// ---- POUs/Lib/Motion/CanOpenAxis/EcCoeSdo/EcCoeSdo_Par_Write_typ.TcDUT
TYPE EcCoeSdo_Par_Write_typ : 	
	STRUCT  (*parameter structure*)
		
        nSubIndex       : BYTE; 
        nIndex          : WORD;
        pSrcBuf         : POINTER TO DWORD; 
        cbBufLen        : UDINT; 
        tTimeout        : TIME := DEFAULT_ADS_TIMEOUT ;

	END_STRUCT
END_TYPE

// ---- POUs/Lib/Motion/CanOpenAxis/EcCoeSdo/EcCoeSdo_Status_typ.TcDUT
TYPE EcCoeSdo_Status_typ : 	
	STRUCT 
		Done : BOOL;
		Busy : BOOL;
		CommandAborted : BOOL;
		Active : BOOL ;
	END_STRUCT
END_TYPE

// ---- POUs/Lib/Motion/CanOpenAxis/eHomingMethods.TcDUT
{attribute 'qualified_only'}
{attribute 'strict'}
TYPE eHomingMethods :
(
	HarsrStopPosDir					:= -2,
	HarsrStopNegDir					:= -1,
	RlsAndIndexPulse 				:= 1,
	FlsAndIndexPulse 				:= 2,
	PositiveSwAndIndexPulse 		:= 3,
	ForwardOnPosSwAndIndexPulse 	:= 4,
	ForwardNegativeSwAndIndexPulse 	:= 5,
	ReverseNegativeSwAndIndexPulse 	:= 6,
	ReverseOnSwAndIndexPulse 		:= 7,
	ForwardOnSwAndIndexPulse 		:= 8,
	ReverseOnPosSwRLSAndIndexPulse	:= 9,
	ForwardOnNegSwAndIndexPulse 	:= 10,
	ForwardOnNegSwAndRLS		 	:= 11,
	ReverseOnPosFLSSwAndIndexPulse	:= 12,
	ForwardOnPosSwRlsAndIndexPulse 	:= 13,
	ReverseOnNegSwRlsAndIndexPulse 	:= 14,
	Reserve1						:= 15,
	Reserve2 						:= 16,
	RlsOnly							:= 17,
	FlsOnly							:= 18,
	ReverseOnNegSw				 	:= 19,
	ForwardOnPosSw					:= 20,
	ForwardOnNegSw					:= 21,
	ReverseOnPosSw				 	:= 22,
	ReverseOnNegFLS				 	:= 23,
	ForwardOnPosFLS					:= 24,
	ReverseOnPosFLS					:= 25,
	ForwardOnNegFLS					:= 26,
	ForwardOnNegRLS					:= 27,
	ReverseOnPosRLS					:= 28,
	ForwardOnPosRLS					:= 29,
	ReverseOnNegRLS					:= 30,
	Reserve3						:= 31,
	Reserve4 						:= 32,	
	IndexPulseNegDir   				:= 33,
	IndexPulsePosDir				:= 34,
	HomeAbs							:= 35,
	HomeCurrent						:= 37 
	
);
END_TYPE

// ---- POUs/Lib/Motion/CanOpenAxis/e_Homing_Contol_Word.TcDUT
{attribute 'qualified_only'}
{attribute 'strict'}
TYPE e_Homing_Contol_Word :
(
	SWITCH_ON 				:= 2#1,		
	Enable_VOLTAGE			:= 2#10,
	QUICK_STOP	 			:= 2#100 ,
	ENABLE_OPERATION		:= 2#1000 ,
	HOME_OPERATION_START	:= 2#10000 ,
	RESERVED1				:= 2#100000 ,
	RESERVED2				:= 2#1000000 ,
	FAULT_RESET				:= 2#10000000 ,
	HALT					:= 2#100000000
);
END_TYPE

// ---- POUs/Lib/Motion/CanOpenAxis/e_Homing_Status_Word.TcDUT
{attribute 'qualified_only'}
{attribute 'strict'}
TYPE e_Homing_Status_Word :
(
	READY_FOR_SWITCH_ON		:= 2#1,		
	SWITCHED_ON				:= 2#10,
	OPERATION_ENABLED		:= 2#100 ,
	FAULT					:= 2#1000 ,
	VOLTAGE_ENABLED			:= 2#10000 ,
	QUICK_STOP				:= 2#100000 , //5
	SWITCH_ON_DISABLED		:= 2#1000000 ,//6
	WARNING					:= 2#10000000 ,//7
	MANAFACTURE_SPECIFIC	:= 2#100000000,
	REMOTE					:= 2#1000000000,//9
	TARGET_REACHED			:= 2#10000000000,//10
	INTERNAL_LIMIT_ACTIVE   := 2#100000000000,//11
	HOMING_ATTAINED			:= 2#1000000000000,//12
	HOMING_ERROR			:= 2#10000000000000,//13	
	RESERVED				:= 2#100000000000000//14,15
);
END_TYPE

// ---- POUs/Lib/Motion/CanOpenAxis/Homing_CoE_Ctrl_Paramters_typ.TcDUT
TYPE Homing_CoE_Ctrl_Paramters_typ :
STRUCT
	HomingMethod  : SINT; 
	HomingSWSpeed : UDINT;
	HomingTrSpeed : UDINT; 
	HomingAcc     : UDINT;
	HomingOffset  : DINT;
 
END_STRUCT
END_TYPE

// ---- POUs/Lib/Motion/ErrorHandling_Lib/Eh_ErrorEntry_typ.TcDUT
TYPE Eh_ErrorEntry_typ:
STRUCT
	SourceId		: UDINT;
	SubSourceId		: UDINT;
	ErrorId			: UDINT;
	ErrorText		: STRING(500);
	MotorEvents		: enumMotorEvents;	
END_STRUCT
END_TYPE

// ---- POUs/Lib/Motion/EtherCAT/SDO_RW/Tc2_EtherCAT_typ/EcCoeSdoRead_CMD_typ.TcDUT
TYPE EcCoeSdoRead_CMD_typ :
	STRUCT
		Enable	: BOOL ;
	END_STRUCT
END_TYPE

// ---- POUs/Lib/Motion/EtherCAT/SDO_RW/Tc2_EtherCAT_typ/EcCoeSdoRead_Param_typ.TcDUT
TYPE EcCoeSdoRead_Param_typ :
	STRUCT
		sNetId          : T_AmsNetId; 
        nSlaveAddr      : UINT; 
        nSubIndex       : BYTE; 
        nIndex          : WORD;
		pDstBuf         : POINTER TO DWORD; 
		cbBufLen        : UDINT; 
		tTimeout        : TIME := DEFAULT_ADS_TIMEOUT; 
	END_STRUCT
END_TYPE

// ---- POUs/Lib/Motion/EtherCAT/SDO_RW/Tc2_EtherCAT_typ/EcCoeSdoRead_Status_typ.TcDUT
TYPE EcCoeSdoRead_Status_typ :
	STRUCT
		bBusy           : BOOL;
        bError          : BOOL;
	END_STRUCT
END_TYPE

// ---- POUs/Lib/Motion/EtherCAT/SDO_RW/Tc2_EtherCAT_typ/EcCoeSdoWrite_CMD_typ.TcDUT
TYPE EcCoeSdoWrite_CMD_typ :
	STRUCT
		Enable	: BOOL ;
	END_STRUCT
END_TYPE

// ---- POUs/Lib/Motion/EtherCAT/SDO_RW/Tc2_EtherCAT_typ/EcCoeSdoWrite_Param_typ.TcDUT
TYPE EcCoeSdoWrite_Param_typ :
	STRUCT
		sNetId          : T_AmsNetId; 
        nSlaveAddr      : UINT; 
        nSubIndex       : BYTE; 
        nIndex          : WORD;
        pSrcBuf         : POINTER TO DWORD; 
        cbBufLen        : UDINT; 
        //bExecute        : BOOL;
        tTimeout        : TIME := DEFAULT_ADS_TIMEOUT ;
	END_STRUCT
END_TYPE

// ---- POUs/Lib/Motion/EtherCAT/SDO_RW/Tc2_EtherCAT_typ/EcCoeSdoWrite_Status_typ.TcDUT
TYPE EcCoeSdoWrite_Status_typ :
	STRUCT
		bBusy           : BOOL;
        bError          : BOOL;
	END_STRUCT
END_TYPE

// ---- POUs/Lib/Motion/EtherCAT/SDO_RW/Tc2_EtherCAT_typ/EcSoeRead_CMD_typ.TcDUT
TYPE EcSoeRead_CMD_typ :
	STRUCT
		Enable	: BOOL ;
	END_STRUCT
END_TYPE

// ---- POUs/Lib/Motion/EtherCAT/SDO_RW/Tc2_EtherCAT_typ/EcSoeRead_Param_typ.TcDUT
TYPE EcSoeRead_Param_typ :
	STRUCT
		sNetId          : T_AmsNetId; 
        nSlaveAddr      : UINT; 
        nSubIndex       : BYTE; 
        nIdn            : WORD;
        nElement        : BYTE;
        nDriveNo        : BYTE;
        bCommand        : BOOL;
        pDstBuf         : POINTER TO DWORD; 
        cbBufLen        : UDINT; 
        bExecute        : BOOL;
        tTimeout        : TIME := DEFAULT_ADS_TIMEOUT;
	END_STRUCT
END_TYPE

// ---- POUs/Lib/Motion/EtherCAT/SDO_RW/Tc2_EtherCAT_typ/EcSoeRead_Status_typ.TcDUT
TYPE EcSoeRead_Status_typ :
	STRUCT
		bBusy           : BOOL;
        bError          : BOOL;
	END_STRUCT
END_TYPE

// ---- POUs/Lib/Motion/EtherCAT/SDO_RW/Tc2_EtherCAT_typ/EcSoeWrite_CMD_typ.TcDUT
TYPE EcSoeWrite_CMD_typ :
	STRUCT
		Enable	: BOOL ;
	END_STRUCT
END_TYPE

// ---- POUs/Lib/Motion/EtherCAT/SDO_RW/Tc2_EtherCAT_typ/EcSoeWrite_Param_typ.TcDUT
TYPE EcSoeWrite_Param_typ :
	STRUCT
		sNetId          : T_AmsNetId; 
        nSlaveAddr      : UINT; 
        nIdn            : WORD; 
        nElement        : BYTE;
        nDriveNo        : BYTE;
        pCommand        : BOOL;
        pSrcBuf         : POINTER TO DWORD; 
        cbBufLen        : UDINT; 
        bExecute        : BOOL;
        tTimeout        : TIME := DEFAULT_ADS_TIMEOUT; 
	END_STRUCT
END_TYPE

// ---- POUs/Lib/Motion/EtherCAT/SDO_RW/Tc2_EtherCAT_typ/EcSoeWrite_Status_typ.TcDUT
TYPE EcSoeWrite_Status_typ :
	STRUCT
		bBusy           : BOOL;
        bError          : BOOL;
	END_STRUCT
END_TYPE

// ---- POUs/Lib/Motion/EtherCAT/SDO_RW/Tc2_EtherCAT_typ/Tc2_EtherCAT_Command_axis_typ.TcDUT
TYPE Tc2_EtherCAT_Command_axis_typ : 	
	STRUCT  (*command structure*)
		EcCoeSdoWrite		: EcCoeSdoWrite_CMD_typ ;
		EcCoeSdoRead		: EcCoeSdoRead_CMD_typ ;
		EcSoeRead			: EcSoeRead_CMD_typ ;
		EcSoeWrite			: EcSoeWrite_CMD_typ ;
	END_STRUCT
END_TYPE

// ---- POUs/Lib/Motion/EtherCAT/SDO_RW/Tc2_EtherCAT_typ/Tc2_EtherCAT_Error_typ.TcDUT
TYPE Tc2_EtherCAT_Error_typ :
	STRUCT
		ErrorID : UDINT ;
		ErrorText : STRING[2048];
	END_STRUCT
END_TYPE

// ---- POUs/Lib/Motion/EtherCAT/SDO_RW/Tc2_EtherCAT_typ/Tc2_EtherCAT_Input_typ.TcDUT
TYPE Tc2_EtherCAT_Input_typ : 	
	STRUCT 
		Command 	: Tc2_EtherCAT_Command_axis_typ;
		Parameter 	: Tc2_EtherCAT_Parameter_axis_typ;
	END_STRUCT
END_TYPE

// ---- POUs/Lib/Motion/EtherCAT/SDO_RW/Tc2_EtherCAT_typ/Tc2_EtherCAT_Output_typ.TcDUT
TYPE Tc2_EtherCAT_Output_typ : 	
	STRUCT 
		Status 	: Tc2_EtherCAT_Statuses_typ;
		Error 	: Tc2_EtherCAT_Error_typ;
	END_STRUCT
END_TYPE

// ---- POUs/Lib/Motion/EtherCAT/SDO_RW/Tc2_EtherCAT_typ/Tc2_EtherCAT_Parameter_axis_typ.TcDUT
TYPE Tc2_EtherCAT_Parameter_axis_typ : 	
	STRUCT  (*parameter structure*)
		EcCoeSdoWrite		: EcCoeSdoWrite_Param_typ ;
		EcCoeSdoRead		: EcCoeSdoRead_Param_typ ;
		EcSoeRead			: EcSoeRead_Param_typ ;
		EcSoeWrite			: EcSoeWrite_Param_typ ;
	END_STRUCT
END_TYPE

// ---- POUs/Lib/Motion/EtherCAT/SDO_RW/Tc2_EtherCAT_typ/Tc2_EtherCAT_Statuses_typ.TcDUT
TYPE Tc2_EtherCAT_Statuses_typ :
	STRUCT
		EcCoeSdoWrite 	: EcCoeSdoWrite_Status_typ ;
		EcCoeSdoRead 	: EcCoeSdoRead_Status_typ ;
		EcSoeRead		: EcSoeRead_Status_typ ;
		EcSoeWrite		: EcSoeWrite_Status_typ ;
	END_STRUCT
END_TYPE

// ---- POUs/Lib/Motion/EtherCAT/SDO_RW/Tc2_EtherCAT_typ/Tc2_EtherCAT_typ.TcDUT
TYPE Tc2_EtherCAT_typ :
	STRUCT
		Input	: Tc2_EtherCAT_Input_typ ;
		Output	: Tc2_EtherCAT_Output_typ ;
	END_STRUCT
END_TYPE

// ---- POUs/Lib/Motion/External Libs/Data types/exCONSTANTS_MATH.TcDUT
TYPE exCONSTANTS_MATH :
STRUCT
	/// Kreiszahl PI 
	PI: REAL := 3.1415926535897931;
	/// PI * 2 
	PI2: REAL := 6.2831853071795862;
	/// PI * 4 
	PI4: REAL := 12.566370614359173;
	/// PI / 2 
	PI05: REAL := 1.5707963267949;
	/// PI / 4 
	PI025: REAL := 0.785398163397448;
	/// 1 / PI 
	PI_INV: REAL := 0.318309886183791;
	/// Euler constant e 
	E: REAL := 2.7182818284590451;
	/// 1 / e 
	E_INV: REAL := 0.367879441171442;
	/// Wurzel von 2 
	SQ2: REAL := 1.4142135623731;
	FACTS: ARRAY[0..12] OF DINT := [1, 1, 2, 6, 24, 120, 720, 5040, 40320, 362880, 3628800, 39916800, 479001600];
END_STRUCT
END_TYPE

// ---- POUs/Lib/Motion/External Libs/Data types/exCONSTANTS_PHYS.TcDUT
TYPE exCONSTANTS_PHYS :
STRUCT
	/// Lichtgeschwindigkeit in m/s 
	C: REAL := 299792458.0;
	/// elementarladung in Colomb = A * s 
	E: REAL := 1.60217653E-19;
	/// Erdbeschleunigung in m / s² 
	G: REAL := 9.80665;
	/// absoluter Nullpunkt in °C 
	T0: REAL := -273.15;
	/// Universelle Gaskonstante in J / (mol · K) 
	RU: REAL := 8.314472;
	/// NormalDruck in Pa 
	PN: REAL := 101325.0;
END_STRUCT
END_TYPE

// ---- POUs/Lib/Motion/FailureRport/Motor/enumFailReportControlFailures.TcDUT
//{attribute 'qualified_only'}
//{attribute 'strict'}
TYPE enumFailReportControlFailures :
(
	IllegalMessageReceived		:=0,
	FunctionBlockError	    	:=1,
	DriveNotReadyForCommand		:=2,
	IllegalParameterReceived	:=3,
	CycleTimeViolation			:=4,
	CommunicationErrorWithDrive	:=5,
	InternalTimeout 			:=6
);
END_TYPE

// ---- POUs/Lib/Motion/FailureRport/Motor/enumFailReportFailureType.TcDUT
//{attribute 'qualified_only'}
//{attribute 'strict'}
TYPE enumFailReportFailureType :
(
	NoFailure 			  :=0,
	MotorFailure 		  :=1,
	ControlFailure 		  :=2,
	CalibrationFailure	  :=3,
	PowerFailure		  :=4,
	FunctionalFailureHigh :=5,
	FunctionalFailureLow  :=6,
	ModuleFailure 		  :=8,
	GeneralDriveError	  :=9
);
END_TYPE

// ---- POUs/Lib/Motion/FailureRport/Motor/enumFailReportMotorFailures.TcDUT
//{attribute 'qualified_only'}
//{attribute 'strict'}
TYPE enumFailReportMotorFailures :
(
	PositionError 			:=0,
	SpeedError				:=1,
	HomeNotFound	 		:=2,
	OverCurrent				:=3,
	OverTemperature			:=4,
	FeedbackError		 	:=5,
	GeneralDriveError 		:=6
);
END_TYPE

// ---- POUs/Lib/Motion/FailureRport/Motor/enumFailReportSeverity.TcDUT
//{attribute 'qualified_only'}
//{attribute 'strict'}
TYPE enumFailReportSeverity :
(
	Warning 	:= 0,
	Error		:= 1,
	Critical	:= 2
	
);
END_TYPE

// ---- POUs/Lib/Motion/FailureRport/Motor/enumMotorEvents.TcDUT
{attribute 'qualified_only'}
{attribute 'strict'}
TYPE enumMotorEvents :
(
	NoEvents				:=0,
	MotorPositionError      :=1,
	MotorSpeedError	        :=2,
	MotorHomeNotFound	    :=3,
	MotorOverCurrent	    :=4,
	MotorOverTemp		    :=5,
	MotorFeedBackErr	    :=6,
	MotorGeneralError		:=7,
	MotorStalled			:=8,
	MotorSupplyError		:=9,
	PLCillegalMsg			:=10,
	PLCIllegalParam			:=11,
	DriveNotEnabled		    :=12,
	DriveNotReady           :=13,
	DriveComError           :=14,
	BreakResistorError      :=15
	
	

);
END_TYPE

// ---- POUs/Lib/Motion/FailureRport/Terminal/Group/Terminal_Group_Ctrl_typ.TcDUT
TYPE Terminal_Group_Ctrl_typ : 	
	STRUCT
  
		In : Terminal_Group_Input_typ;
		
		Out : Terminal_Group_Output_typ;
		
	END_STRUCT
END_TYPE

// ---- POUs/Lib/Motion/FailureRport/Terminal/Group/Terminal_Group_Input_typ.TcDUT
TYPE Terminal_Group_Input_typ : 	
	STRUCT 
		Par : Terminal_Group_Parameter_typ;
	END_STRUCT
END_TYPE

// ---- POUs/Lib/Motion/FailureRport/Terminal/Group/Terminal_Group_Monitor_typ.TcDUT
TYPE Terminal_Group_Monitor_typ : 	
	STRUCT  
		SubSysName		: STRING[20];	
	END_STRUCT
END_TYPE

// ---- POUs/Lib/Motion/FailureRport/Terminal/Group/Terminal_Group_Output_typ.TcDUT
TYPE Terminal_Group_Output_typ : 	
	STRUCT  
		Status:  Terminal_Group_Status_typ;
		Monitor: Terminal_Group_Monitor_typ;
	END_STRUCT
END_TYPE

// ---- POUs/Lib/Motion/FailureRport/Terminal/Group/Terminal_Group_Parameter_typ.TcDUT
TYPE Terminal_Group_Parameter_typ : 	
	STRUCT  (*parameter structure*)
		GroupName			: STRING[20];
		GroupID				: USINT;	
		PosForLog			: USINT;
	END_STRUCT
END_TYPE

// ---- POUs/Lib/Motion/FailureRport/Terminal/Group/Terminal_Group_Status_typ.TcDUT
TYPE Terminal_Group_Status_typ : 	
	STRUCT  		
		Active:         BOOL;	
		errorBit:       ULINT; 
		
	END_STRUCT
END_TYPE

// ---- POUs/Lib/Motion/FailureRport/Terminal/Terminal/Terminal_Ctrl_typ.TcDUT
TYPE Terminal_Ctrl_typ : 	
	STRUCT
  
		In : Terminal_Input_typ;
		
		Out : Terminal_Output_typ;
		
	END_STRUCT
END_TYPE

// ---- POUs/Lib/Motion/FailureRport/Terminal/Terminal/Terminal_Input_typ.TcDUT
TYPE Terminal_Input_typ : 	
	STRUCT 
		Par : Terminal_Parameter_typ;
	END_STRUCT
END_TYPE

// ---- POUs/Lib/Motion/FailureRport/Terminal/Terminal/Terminal_Monitor_typ.TcDUT
TYPE Terminal_Monitor_typ : 	
	STRUCT  
		SubSysName		: STRING[20];	
	END_STRUCT
END_TYPE

// ---- POUs/Lib/Motion/FailureRport/Terminal/Terminal/Terminal_Output_typ.TcDUT
TYPE Terminal_Output_typ : 	
	STRUCT  
		Status:  Terminal_Status_typ;
		Monitor: Terminal_Monitor_typ;
	END_STRUCT
END_TYPE

// ---- POUs/Lib/Motion/FailureRport/Terminal/Terminal/Terminal_Parameter_typ.TcDUT
TYPE Terminal_Parameter_typ : 	
	STRUCT  (*parameter structure*)
		Name				: STRING[30] :=  'Empty';
		ModuleID			: UINT;		
		PosForLog			: USINT;
	END_STRUCT
END_TYPE

// ---- POUs/Lib/Motion/FailureRport/Terminal/Terminal/Terminal_Status_typ.TcDUT
TYPE Terminal_Status_typ : 	
	STRUCT  
		TerminalState:  UDINT;
		Active:         BOOL;	
		Fault:          BOOL;
	END_STRUCT
END_TYPE

// ---- POUs/Lib/Motion/SercosAxis/SercosDrive_Ctrl_Adr_typ.TcDUT
TYPE SercosDrive_Ctrl_Adr_typ :
STRUCT
	//output
	ControlWord      : WORD;
	DriveError:       WORD;
	Diagnostic:       WORD;	
END_STRUCT
END_TYPE

// ---- POUs/Lib/ProgramBasic/LocalEvent_Typ.TcDUT
TYPE LocalEvent_Typ :
STRUCT
	EventHeader:EventHeader_Typ;
	EventParameters:EventParam_Typ;
	rEvent : REFERENCE TO EventHelper;
//	flowId:DINT;
END_STRUCT
END_TYPE

// ---- POUs/Lib/Signal/E_LutMode.TcDUT
{attribute 'qualified_only'}
{attribute 'strict'}
TYPE E_LutMode :
(
	eDisabled:= 0,
	ePhisicalToAnalog:= 1,
	eAnalogToPhisical:= 2
);
END_TYPE

// ---- POUs/Lib/Signal/ST_LookUpTableParam.TcDUT
TYPE ST_LookUpTableParam	 :
STRUCT
	arrPhisical:	ARRAY[0..40] OF LREAL;
	arrAnalog:		ARRAY[0..40] OF LINT;
	eLutMode:		E_LutMode;			
END_STRUCT
END_TYPE

// ---- POUs/Lib/System/CmdQueue/DUTs/DelayInfo_typ.TcDUT
TYPE DelayInfo_typ :
STRUCT	
	RequestId : UDINT;
	GroupId : UDINT;
	DelayType : eDelayType;
	DelayValue : ULINT; // ms or microns
	pExecuted : POINTER TO BOOL; // need to be persistant
	PrivateInfo : PVOID;
	Executed : BOOL;
	LagError : UDINT; // ms or microns
END_STRUCT
END_TYPE

// ---- POUs/Lib/System/CmdQueue/DUTs/eDelayType.TcTLEO
{attribute 'qualified_only'}
{attribute 'strict'}
TYPE eDelayType :
(
	Immediate := 0,
	DelayByTimer := 1,
	DelayByPos := 2
);
END_TYPE

// ---- GVLs/AxesList.TcGVL
//{attribute 'qualified_only'}
VAR_GLOBAL
	gWebAxes:		WebAxes_typ;	
END_VAR

// ---- GVLs/Consts.TcGVL
//{attribute 'qualified_only'}
VAR_GLOBAL CONSTANT
CONST_ZERO :DINT :=0;	





END_VAR

VAR_GLOBAL CONSTANT

// States		
	MACHINE_RUN_INIT:						INT:=0;
	MACHINE_GRIPPER_START_POSITION:			INT:=11;
	MACHINE_GRIPPER_EXCTRACT:				INT:=12;
	MACHINE_GRIPPER_OPEN:					INT:=13;
	MACHINE_GRIPPER_CLOSE:					INT:=14;
	MACHINE_GRIPPER_RETRACT:				INT:=15;
	
	MACHINE_GRIPPER_END_POSITION:			INT:=17;
	MACHINE_ENABLE_TENSION:					INT:=18;	
	//MACHINE_FRIPPER_WAIT_POSITION:			INT:=19;	
	
	MACHINE_WAIT_DANCER_FULL:				INT:=21;
	
	
	MACHINE_COLD_CUT_VALVE_OPEN:				INT:=10;
	MACHINE_WELD_VALVE_OPEN:					INT:=20;	
	MACHINE_HEATER_ON:							INT:=30;	
	MACHINE_HEATER_OFF:							INT:=40;
	MACHINE_VALVE_CLOSE:						INT:=50;	
	
	MACHINE_OUT_GRIPPER_START_POSITION:			INT:=60;
	MACHINE_OUT_GRIPPER_CLAMP:					INT:=61;
	MACHINE_OUT_GRIPPER_END_POSITION:			INT:=62;	
	
	MACHINE_CUT_WEB:							INT:=63;

	MACHINE_DONE:							INT:=100;	



END_VAR

// ---- GVLs/GVL.TcGVL
//{attribute 'qualified_only'}
VAR_GLOBAL
gMachineCtrl: Ctrl_Typ;
	
FB_Machine_Ctrl:FB_Machine_Ctrl;
FB_Machine_Run:FB_Machine_Run;
FB_Mechinit:FB_Mechinit;
FB_OFF:FB_OFF;
FB_Mechinit_Output:FB_MechinitOutput;

FB_RW_Ctrl:FB_RW_Ctrl;
RwInverter :FB_INV;


//WebHandling
	UW_1_AxisFB			: Beck5xxxAxis_FB;
	UW_1_MultiAxisFB	: MultiAxis_FB;
	UW_1_CyclicAxisFB	: CyclicAxis_FB;
	
	UW_2_AxisFB			: Beck5xxxAxis_FB;
	UW_2_MultiAxisFB	: MultiAxis_FB;
	UW_2_CyclicAxisFB	: CyclicAxis_FB;	
	
	Output_AxisFB		: ElmoBasicAxis_FB;
//	Uutput_MultiAxisFB	: MultiAxis_FB;
//	Uutput_CyclicAxisFB	: CyclicAxis_FB;
	
	UwVmaster_AxisFB		: CoE_BasicAxis_FB;
	
	//UW_MotorFailureReportFB 		: MotorFailureReport_FB;
	//UWMaster_MotorFailureReportFB 	: MotorFailureReport_FB;
	
END_VAR

// ---- GVLs/Persist.TcGVL
//{attribute 'qualified_only'}
VAR_GLOBAL  PERSISTENT 
    PersistentStruct:Persistent_Typ;
END_VAR

// ---- POUs/Lib/Logging/logLib/GVL_1.TcGVL
//{attribute 'qualified_only'}
VAR_GLOBAL CONSTANT
	MAX_COUNT_LOG_PARAM		: USINT := 5;	(*Maximum parameters index in log message variable data (from 0)*)
	LOCAL_ARRAY_LENGTH		: UINT := 32;	(* power oof 2 : The length of local (per task) array*)
	MAX_MEMBERS_TO_WRITE	: USINT := 8;
	GLOBAL_ARRAY_LENGTH		: UINT := 4*1024;(* power oof 2 : The length of global array*)
	LOG_TPL					: USINT := 0;
	LOG_MAIN_MOTOR			: USINT := 1;
	ENUM_OF_LAST_TASK		: USINT := 1;
	LOG_MSG_CATEGORY_LENGTH	: UINT := 10;
	LOG_MSG_TEXT_LENGTH		: USINT := 210;	(*The maximal length of log text *)
END_VAR

VAR_GLOBAL

END_VAR

// ---- POUs/Lib/Logging/PLC_ClientComm/UDP_Comm/PcComm/PcComm.TcGVL
//{attribute 'qualified_only'}
VAR_GLOBAL
	LogGlobalArray : LogGlobalArrayObj;	
END_VAR

// ---- POUs/Lib/Motion/External Libs/Global Variables/exConstants.TcGVL
{attribute 'Tc2GvlVarNames' := ''}
VAR_GLOBAL CONSTANT
	STRING_LENGTH: INT := 250;
	LIST_LENGTH: INT := 250;
END_VAR

// ---- POUs/Lib/Motion/External Libs/Global Variables/exGlobale_Variablen.TcGVL
{attribute 'Tc2GvlVarNames' := ''}
VAR_GLOBAL
	MATH: exCONSTANTS_MATH;
	PHYS: exCONSTANTS_PHYS;

END_VAR

// ---- POUs/MAIN.TcPOU
PROGRAM MAIN
VAR

init:BOOL;

uw1_Toque AT %I* 	: INT;
uw1_Position AT %I* 	: DINT;
TriggerOff:Trigger;
TriggerEM_Button:Trigger;

BuzzerTimer:TON;
END_VAR


IF init =FALSE THEN
	init:=TRUE;
	ACT_Init_param();
END_IF

ACT_Emergency();

ACT_IO();

ACT_fbCall();

ACT_Buzzer();

ACTION ACT_Buzzer:

BuzzerTimer.IN:= gMachineCtrl.IO.Out.PressDown OR gMachineCtrl.IO.Out.ColdCutPistonDown;
BuzzerTimer.PT:= T#3S;
BuzzerTimer();
IF gMachineCtrl.IO.Out.PressDown
AND  BuzzerTimer.Q = FALSE THEN
	gMachineCtrl.IO.Out.Buzzer := TRUE;
ELSE
	gMachineCtrl.IO.Out.Buzzer := FALSE;
END_IF
END_ACTION

ACTION ACT_Emergency:

IF gMachineCtrl.Cmd.EmStop THEN
	//FB_Machine_Ctrl.ResetCycle:=TRUE;
	//gMachineCtrl.Cmd.EmStop:=FALSE;
	
	gMachineCtrl.Cmd.SwitchOn:=FALSE;
END_IF
IF TriggerOff.EDGENEG(gMachineCtrl.Cmd.SwitchOn) THEN
	gMachineCtrl.Cmd.EmStop:=TRUE;
END_IF

IF TriggerEM_Button.EDGEPOS(gMachineCtrl.Cmd.EmStop) THEN
	gMachineCtrl.Cmd.EmStop:=TRUE;
END_IF
END_ACTION

ACTION ACT_fbCall:



RwInverter(
	//Set_Vel_Link:=gUVCtrl.Input.Par.UV_Inverter_Set_Speed , 
	//INV_Enable:=gUVCtrl.Input.Cmd.UV_Inverter_Run , 
	//HWlink:=gMachineCtrl.IO.RwInverter,
	ctrl:=gMachineCtrl.RwInverter,
	//ResetError:= , 
	MasterNetId:= , 
	nSlaveAddr:= , 
	nSubIndex:= , 
	nIndex:= , 
	//Actual_Vel_Link=>gUVCtrl.Output.Status.UV_Inverter_Actual_Speed , 
	Error=> , 
	ErrorCode=> , 
	Inv_Status=> );


	
FB_OFF.Ctrl_ref 			REF= gMachineCtrl;
FB_OFF.FB_Machine_Run_ref 	REF= FB_Machine_Run;
FB_OFF.FB_Mechinit_ref 		REF= FB_Mechinit;
FB_OFF();	
	
FB_Machine_Ctrl.Ctrl_ref 				REF= gMachineCtrl;
FB_Machine_Ctrl.FB_Machine_Run_ref 		REF= FB_Machine_Run;
FB_Machine_Ctrl.FB_Mechinit_ref 		REF= FB_Mechinit;
FB_Machine_Ctrl.FB_MechinitOutput_ref  	REF= FB_Mechinit_Output;
FB_Machine_Ctrl.FB_OFF_ref				REF= FB_OFF;
FB_Machine_Ctrl();

FB_Machine_Run.Ctrl_ref 		REF= gMachineCtrl;
FB_Machine_Run.FB_RW_Ctrl_ref	REF= FB_RW_Ctrl;
FB_Machine_Run();


FB_Mechinit.Ctrl_ref	REF= gMachineCtrl;
FB_Mechinit();


FB_Mechinit_Output.Ctrl_ref	REF= gMachineCtrl;
FB_Mechinit_Output();

//FB_RW_Ctrl.Ctrl_ref REF= gMachineCtrl;
//FB_RW_Ctrl();
END_ACTION

ACTION ACT_Init_param:

//	Dancer fill speed
gMachineCtrl.Parameters.DancerFillSpeed:= 90000;//[mil deg/sec]

gMachineCtrl.Parameters.NumberOfCycles:= 1;

//Motor Parmeters
//gMachineCtrl.Parameters.MotorVelocity:=600;//[rpm]
gMachineCtrl.Parameters.DistanceToMove:=1000;//[mm]


gMachineCtrl.Parameters.WebLinarSpeed:=350;//[mm/sec]
gMachineCtrl.Parameters.WebLinarSpeedSlow:=250;//[mm/sec]

gMachineCtrl.Parameters.UW_1_Param.ForcedDiameter:=400;//[mm/sec]
gMachineCtrl.Parameters.UW_2_Param.ForcedDiameter:=400;//[mm/sec]

gMachineCtrl.Parameters.UW_1_Param.SetTension := 150;
gMachineCtrl.Parameters.UW_2_Param.SetTension := 150;

gMachineCtrl.Parameters.UW_1_Param.kp:=0.1;
gMachineCtrl.Parameters.UW_1_Param.TN:=T#0MS;

gMachineCtrl.Parameters.UW_2_Param.kp:=0.1;
gMachineCtrl.Parameters.UW_2_Param.TN:=T#0MS;

gMachineCtrl.Parameters.UW_1_Param.kpMove:=1;
gMachineCtrl.Parameters.UW_1_Param.TNMove:=T#0MS;

gMachineCtrl.Parameters.UW_2_Param.kpMove:=1;
gMachineCtrl.Parameters.UW_2_Param.TNMove:=T#0MS;

//Output
gMachineCtrl.Parameters.OutGripperEndPosition :=1800;//mm
gMachineCtrl.Parameters.OutGripperHomeVelocity:=75;//mm
gMachineCtrl.Parameters.OutGripperProcessVelocity:=1000;//mm
END_ACTION

ACTION ACT_IO:


//IO
gMachineCtrl.IO.In.PrimeryPressFeedback(
	SimFlag:= gMachineCtrl.Simulation);
	
gMachineCtrl.IO.In.SeconderyPressFeedbak(
	SimFlag:= gMachineCtrl.Simulation);
	
gMachineCtrl.IO.In.E_StopPressed := NOT(gMachineCtrl.IO.In.E_StopPressedRaw);

gMachineCtrl.IO.In.UW_1_DancerFull :=NOT( gMachineCtrl.IO.In.UW_1_DancerFullRaw);
gMachineCtrl.IO.In.UW_2_DancerFull :=NOT( gMachineCtrl.IO.In.UW_2_DancerFullRaw);	

gMachineCtrl.IO.In.UW_1_DancerEmpety :=NOT( gMachineCtrl.IO.In.UW_1_DancerEmpetyRaw);
gMachineCtrl.IO.In.UW_2_DancerEmpety :=NOT( gMachineCtrl.IO.In.UW_2_DancerEmpetyRaw);	

gMachineCtrl.IO.Out.Output_GripperOpen:= NOT (gMachineCtrl.IO.Out.Output_GripperClose);
END_ACTION

END_PROGRAM

// ---- POUs/Lib/Trigger.TcPOU
FUNCTION_BLOCK FINAL Trigger
VAR_INPUT
END_VAR
VAR_OUTPUT
END_VAR
VAR
	rTrig : R_TRIG ;
	ftrig : F_TRIG ;
END_VAR

METHOD PUBLIC EDGENEG : BOOL
VAR_INPUT
	input : BOOL ;
END_VAR

fTrig.CLK := input ;
fTrig();

EDGENEG := fTrig.Q ;
END_METHOD

METHOD PUBLIC EDGEPOS : BOOL
VAR_INPUT
	input : BOOL ;
END_VAR

rTrig.CLK := input ;
rTrig();

EDGEPOS := rTrig.Q ;
END_METHOD

METHOD ONE_SHOT : BOOL
VAR_INPUT
	input : BOOL ;
END_VAR
rTrig.CLK := input ;
rTrig();

fTrig.CLK := input ;
fTrig();

ONE_SHOT := rTrig.Q OR fTrig.Q;
END_METHOD

END_FUNCTION_BLOCK

// ---- POUs/App/FB_OFF.TcPOU
FUNCTION_BLOCK FB_OFF EXTENDS CycleHandleFB
VAR_INPUT
	Ctrl_ref:			REFERENCE TO Ctrl_Typ;
	FB_RW_Ctrl_ref:			REFERENCE TO FB_RW_Ctrl;
	FB_Machine_Run_ref:		REFERENCE TO FB_Machine_Run;
	FB_Mechinit_ref:		REFERENCE TO FB_Mechinit;

	
END_VAR
VAR_OUTPUT
END_VAR
VAR
	MethInitDone:		BOOL;
END_VAR

VAR CONSTANT
// States are global
		
	OFF_INIT:			INT:=0;
	OFF_STOP_MOTOR:		INT:=5;
	OFF_GEAR_OUT:		INT:=6;
	OFF_MOTOR:			INT:=10;
	OFF_RESET_CYCLES:	INT:=20;
	OFF_RESET_IO:	INT:=30;
	OFF_DONE:			INT:=100;
END_VAR



IF NOT MethInitDone THEN
	MethInitDone	:= Meth_Init();
END_IF

IF  THIS^.CMD.Pause = FALSE THEN
	
	//-----------------------------
	//State Machine
	//-----------------------------
	CASE THIS^.StepNo OF
		OFF_INIT:
			IF THIS^.StepOneShotTrig THEN
				THIS^.Monitoring.StepMessage	:= 'Init: Start.';
				THIS^.Delay(IN:=FALSE);
			ELSIF Meth_Enable(TRUE) THEN
				THIS^.StepNo	:= 	OFF_RESET_IO;
			END_IF
			
			OFF_RESET_IO:
				IF THIS^.StepOneShotTrig THEN
					THIS^.Monitoring.StepMessage	:= 'Rest all IO';
				ELSIF Meth_Rest_IO() THEN
					THIS^.StepNo	:= 	OFF_GEAR_OUT;
				END_IF			
			
			OFF_GEAR_OUT:
				IF THIS^.StepOneShotTrig THEN
					THIS^.Monitoring.StepMessage	:= 'Gear Out';
					THIS^.Meth_GearOut(FALSE);
				ELSIF Meth_GearOut(TRUE) THEN
					THIS^.StepNo	:= 	OFF_STOP_MOTOR;
				END_IF					
				
			OFF_STOP_MOTOR:
				IF THIS^.StepOneShotTrig THEN
					THIS^.Monitoring.StepMessage	:= 'Stop Motors';
					THIS^.Meth_StopMotors(FALSE);
				ELSIF Meth_StopMotors(TRUE) THEN
					THIS^.StepNo	:= 	OFF_MOTOR;
				END_IF					
				
			OFF_MOTOR:
				IF THIS^.StepOneShotTrig THEN
					THIS^.Monitoring.StepMessage	:= 'Switch Motors Off';
					THIS^.Meth_SwitchOff(FALSE);
				ELSIF Meth_SwitchOff(TRUE) THEN
					THIS^.StepNo	:= 	OFF_RESET_CYCLES;
				END_IF		

			OFF_RESET_CYCLES:
				IF THIS^.StepOneShotTrig THEN
					THIS^.Monitoring.StepMessage	:= 'Rest all cycles';
				ELSIF Meth_ResatAllCycles() THEN
					THIS^.StepNo	:= 	OFF_DONE;
				END_IF				
				
					
				
			OFF_DONE:
				IF THIS^.StepOneShotTrig THEN
					THIS^.Monitoring.StepMessage	:= 'OFF cycle Done';
				ELSIF Meth_Done(TRUE) THEN
					THIS^.StepNo	:= 	OFF_INIT;
				END_IF					
				
		END_CASE
	
	ELSE
		THIS^.Monitoring.StepMessage:= 'Pause';
		
		IF THIS^.Status.Fault = TRUE THEN
		//IF Meth_EmStop(TRUE) THEN
				THIS^.CMD.ResetCycle	:= TRUE;		// Reset the all state machine to start point
		//END_IF
			
		END_IF
		
	END_IF
	
	THIS^.Delay();
	THIS^.CH_Logic();
	
	// Reset Meth_EmStop when at Init State
	IF THIS^.Pause = FALSE THEN
		//Meth_EmStop(FALSE);
	END_IF

METHOD PRIVATE Meth_Done : BOOL
VAR_INPUT
	Execute: 	BOOL;
END_VAR


	//THIS^.Monitoring.StepMessage			:= 'Press 1 engage';
	//THIS^.Monitoring.Error_Text				:= 'Press 1 engage Fail';
	//THIS^.CMD.Deacivate_Sequence_Time_Out	:= TRUE;	// Disable time out to the all sequence
	//THIS^.CMD.DeactivateStepTimeOut			:= TRUE;	// Disable time out to the actual step
	//THIS^.Parameter.TimeOut					:= T#5S;

	THIS^.Status.Done		:= TRUE;
	THIS^.Status.Running	:= FALSE;									
	Meth_Done	:= TRUE;
END_METHOD

METHOD PRIVATE Meth_Enable : BOOL
VAR_INPUT
	Execute: 	BOOL;
END_VAR


IF THIS^.CMD.Start THEN
	
	THIS^.Monitoring.StepMessage			:= 'Start';
	THIS^.Monitoring.Error_Text				:= 'Start Fail';
	THIS^.CMD.Deacivate_Sequence_Time_Out	:= TRUE;	// Disable time out to the all sequence
	THIS^.CMD.DeactivateStepTimeOut			:= TRUE;	// Disable time out to the actual step
	THIS^.Parameter.TimeOut					:= T#0.5S;

	THIS^.CMD.Start			:= FALSE;
	THIS^.Status.Done		:= FALSE;
	THIS^.Status.Running	:= TRUE;
	
	// Reset Commands and Statuses												
	
	Meth_Enable	:= TRUE;
END_IF
END_METHOD

METHOD Meth_GearOut : BOOL
VAR_INPUT
	Execute: 	BOOL;
END_VAR
VAR_INST	
	ExecuteTrig: 	Trigger;	
END_VAR
IF ExecuteTrig.EDGEPOS(Execute) THEN
	Meth_GearOut	:= FALSE;
	THIS^.SubStepNo:= 	1;	
END_IF

IF ExecuteTrig.EDGENEG(Execute) THEN
	Meth_GearOut	:=	FALSE;
END_IF

CASE THIS^.SubStepNo OF
	   
	1:
	
		IF (gWebAxes.UW_1.Crtl.Basic_axis.Output.Status.AxisStatus.SynchronizedMotion = TRUE) THEN
			THIS^.Monitoring.StepMessage	:= 'Set Gear out command UW1';							
			gWebAxes.UW_1.Crtl.MultiAxis.Input.Command.GearInMultiMaster.DisengageSlave	:= TRUE;
			THIS^.SubStepNo	:= 2;	
		ELSE
			THIS^.Monitoring.StepMessage	:= 'UW1 not synchronized, continue';	
			THIS^.SubStepNo	:= 2;				
		END_IF	
			
	
	2:	
		IF (gWebAxes.UW_2.Crtl.Basic_axis.Output.Status.AxisStatus.SynchronizedMotion = TRUE) THEN
			THIS^.Monitoring.StepMessage	:= 'Set Gear out command UW2';							
			gWebAxes.UW_2.Crtl.MultiAxis.Input.Command.GearInMultiMaster.DisengageSlave	:= TRUE;
			THIS^.SubStepNo	:= 3;	
		ELSE
			THIS^.Monitoring.StepMessage	:= 'UW2 not synchronized, continue';	
			THIS^.SubStepNo	:= 3;				
		END_IF	
		
	3:	
		THIS^.Monitoring.StepMessage:= 'Wait for Gear out UW 1+2';
									
		IF  gWebAxes.UW_1.Crtl.Basic_axis.Output.Status.AxisStatus.SynchronizedMotion = FALSE
		AND gWebAxes.UW_2.Crtl.Basic_axis.Output.Status.AxisStatus.SynchronizedMotion = FALSE THEN
			Meth_GearOut:=TRUE;
		END_IF	

							
END_CASE
END_METHOD

METHOD Meth_Init :BOOL
VAR_INPUT
END_VAR
//resets


Meth_Init:=TRUE;
END_METHOD

METHOD Meth_ResatAllCycles : BOOL
VAR_INPUT
END_VAR

FB_Machine_Run_ref.ResetCycle	 :=TRUE;
FB_Mechinit_ref.ResetCycle		 :=TRUE;


Meth_ResatAllCycles:=TRUE;
END_METHOD

METHOD Meth_Rest_IO : BOOL
VAR_INPUT
	
END_VAR

Ctrl_ref.IO.Out.HeaterOn := FALSE;
gMachineCtrl.IO.Out.GripperRetract:=FALSE;
gMachineCtrl.IO.Out.GripperOpen:=FALSE;

gMachineCtrl.IO.Out.ExternalNipMotor:=FALSE;

gMachineCtrl.IO.Out.Output_GripperClose:=FALSE;

gMachineCtrl.IO.Out.Buzzer	:=FALSE;

gMachineCtrl.IO.Out.ColdCutPistonDown:=FALSE;	

Meth_Rest_IO:=TRUE;
END_METHOD

METHOD Meth_StopMotors : BOOL
VAR_INPUT
	Execute: 	BOOL;
END_VAR
VAR_INST	
	ExecuteTrig: 	Trigger;	
END_VAR
IF ExecuteTrig.EDGEPOS(Execute) THEN
	Meth_StopMotors	:= FALSE;
	THIS^.SubStepNo:= 	1;	
END_IF

IF ExecuteTrig.EDGENEG(Execute) THEN
	Meth_StopMotors	:=	FALSE;
END_IF

CASE THIS^.SubStepNo OF
	   
	1:
		THIS^.Monitoring.StepMessage:= 'Stop Motors';
		
		gWebAxes.UW_1.Crtl.Basic_axis.Input.Parameter.Acceleration := 	10000000;
		gWebAxes.UW_1.Crtl.Basic_axis.Input.Parameter.Deceleration := 	10000000;		
		gWebAxes.UW_1.Crtl.Basic_axis.Input.Command.Stop :=		TRUE;
		
		gWebAxes.UW_2.Crtl.Basic_axis.Input.Parameter.Acceleration := 	10000000;
		gWebAxes.UW_2.Crtl.Basic_axis.Input.Parameter.Deceleration := 	10000000;		
		gWebAxes.UW_2.Crtl.Basic_axis.Input.Command.Stop :=		TRUE;		
		
		gWebAxes.Output.Crtl.Basic_axis.Input.Parameter.Acceleration := 	10000;//[mm
		gWebAxes.Output.Crtl.Basic_axis.Input.Parameter.Deceleration := 	10000;		
		gWebAxes.Output.Crtl.Basic_axis.Input.Command.Stop :=		TRUE;		
						
				
								
		THIS^.SubStepNo	:= 2;		
			
	
	2:	
		THIS^.Monitoring.StepMessage:= 'Wait for standstill UW 1';
									
		IF gWebAxes.UW_1.Crtl.Basic_axis.Output.Status.AxisStatus.StandStill
		OR gWebAxes.UW_1.Crtl.Basic_axis.Output.Status.AxisStatus.Disabled THEN
			THIS^.SubStepNo	:= 3 ;
		END_IF
		
	3:	
		THIS^.Monitoring.StepMessage:= 'Wait for standstill UW 2';
									
		IF gWebAxes.UW_1.Crtl.Basic_axis.Output.Status.AxisStatus.StandStill
		OR  gWebAxes.UW_2.Crtl.Basic_axis.Output.Status.AxisStatus.Disabled THEN
			THIS^.SubStepNo	:= 4 ;
		END_IF	

	4:	
		THIS^.Monitoring.StepMessage:= 'Wait for standstill Output';
									
		IF gWebAxes.Output.Crtl.Basic_axis.Output.Status.AxisStatus.StandStill
		OR  gWebAxes.Output.Crtl.Basic_axis.Output.Status.AxisStatus.Disabled THEN
			//THIS^.SubStepNo	:= 4 ;
			Meth_StopMotors:=TRUE;
		END_IF								
END_CASE
END_METHOD

METHOD Meth_SwitchOff : BOOL
VAR_INPUT
	Execute: 	BOOL;
END_VAR
VAR_INST
	ExecuteTrig: 	Trigger;
END_VAR


IF ExecuteTrig.EDGEPOS(Execute) THEN
	Meth_SwitchOff:=	FALSE;
	THIS^.SubStepNo:= 	1;	
END_IF

IF ExecuteTrig.EDGENEG(Execute) THEN
	Meth_SwitchOff:=	FALSE;
END_IF

CASE THIS^.SubStepNo OF
	(* Power ON*)
	1:
		THIS^.Monitoring.StepMessage	:= 'Power OFF';								
		gWebAxes.UW_1.Crtl.Basic_axis.Input.Command.Power		:= FALSE;
		gWebAxes.UW_2.Crtl.Basic_axis.Input.Command.Power		:= FALSE;	
		gWebAxes.Output.Crtl.Basic_axis.Input.Command.Power		:= FALSE;
		
		THIS^.SubStepNo:= 2;		
	
	2:	
		THIS^.Monitoring.StepMessage:= 'Wait for Disabled UW 1';
									
		IF gWebAxes.UW_1.Crtl.Basic_axis.Output.Status.AxisStatus.Disabled THEN
			THIS^.SubStepNo	:= 3 ;
		END_IF
		
	3:	
		THIS^.Monitoring.StepMessage:= 'Wait for Disabled UW 2';
									
		IF gWebAxes.UW_2.Crtl.Basic_axis.Output.Status.AxisStatus.Disabled  THEN
			THIS^.SubStepNo	:= 4 ;
		END_IF	
	4:	
		THIS^.Monitoring.StepMessage:= 'Wait for Disabled Output';
									
		IF gWebAxes.Output.Crtl.Basic_axis.Output.Status.AxisStatus.Disabled  THEN
			Meth_SwitchOff	:= TRUE;
		END_IF		
		
							
END_CASE
END_METHOD

END_FUNCTION_BLOCK

// ---- POUs/Lib/CH Obj/CycleHandleFB.TcPOU
FUNCTION_BLOCK  CycleHandleFB 
VAR_IN_OUT

END_VAR

VAR_INPUT
	//pFlowID: 			POINTER TO DINT :=ADR(DummyFlowID) ;
	SetEvent:			BOOL;
		
END_VAR
VAR_OUTPUT
	//Error 				: Error_Handler_typ;
END_VAR
VAR 
	// ErrorReportStruct 	:  FailureReport_Typ;	

	CMD					: Basic_cycle_CMD_typ ;
	Monitoring			: Basic_cycle_Mon_typ ;
	Status				: Basic_cycle_Status_typ ;
	Parameter			: Basic_cycle_Param_typ ;
	AtReady				: BOOL;
	Delay 				: TON ;
	StepOneShotTrig		: BOOL;
	LogMsg_0 			: LogMsg ;
	//fbClearFaultHandler_0 : fbClearFaultHandler;
	ResetError 			: R_TRIG;
	rTrigCycleDone 		: R_TRIG;
	fTrigCycleRunning 	: F_TRIG;
	rTrigCycleStart		: R_TRIG;	
	Init_trig 			: R_TRIG;
	ResetFaultTrig 		: R_TRIG;
	ResetAllTrig 		: R_TRIG;
	ResumeAllTrig 		: R_TRIG;
	LastStepMessage 	: STRING[100];
	LastStepNo 			: DINT;
	LastSubStepNo		: DINT ;
	TimeOutFault		: BOOL;
	CycleTIME 			: TON;
	StepTimerTOut 		: TON;
	SubStepTimerTOut 	: TON;
	ErrorAcknowledge 	: BOOL;
	Triger1 			: Trigger ;
	Triger2 			: Trigger ;
	Triger3 			: Trigger ;
	Triger4 			: Trigger ; 
	Triger5 			: Trigger ; 

	DummyFlowID			: DINT :=0;
	//fbCHPrgmBasic 		: FB_PrgmBasic;

	//rEvent : 			REFERENCE TO EventHelper;
	//EventHeader:		EventHeader_Typ;
	//EventParameters:	EventParam_Typ;	
END_VAR

METHOD PROTECTED CH_Logic : BOOL
VAR_STAT
	EventSent: 			BOOL;
END_VAR
VAR
	stenNomForLog	: DINT;
END_VAR

	IF CMD.LogMsgInit THEN      
		CMD.LogMsgInit := FALSE ;
		fnLogMsgInit(ADR(LogMsg_0), Parameter.ThreadName, ADR(LogGlobalArray), ADR(Parameter.PosForLog));
		LogMsg_0.Enable:= 		TRUE;
		CMD.EnableStateLogging:= TRUE;
		Parameter.ExternalLogType := LOG_INFO ;
	END_IF

	// Write state name for every change of Step Message
	IF (Monitoring.StepMessage) <> (LastStepMessage) THEN
		LastStepMessage := Monitoring.StepMessage ;
		// fnLogMsg(ADR(LogMsg_0), LOG_INFO, CONCAT(CONCAT(Parameter.CHName,', State = %d, FlowID = %d '),Monitoring.StepMessage),LastStepNo,pFlowID^,0);	
		IF CMD.EnableStateLogging THEN
			IF (Parameter.StepMessageIsForNewState) THEN
				Parameter.StepMessageIsForNewState	:= FALSE;
				stenNomForLog	:= StepNo;
			ELSE
				stenNomForLog	:= LastStepNo;
			END_IF
			fnLogMsg(ADR(LogMsg_0), LOG_INFO, CONCAT(CONCAT(CONCAT(Parameter.CHName, ', '),Monitoring.StepMessage),', State = %d.'), stenNomForLog,0,0);	
		END_IF
	END_IF
	
	

				
	//Update Step Num for Visu
	IF Triger1.EDGEPOS(Monitoring.LastStep <> Monitoring.StepNo) THEN 
		Monitoring.Visu_StepNo := LastStepNo ;
	ELSIF Status.CycleStuck AND NOT CMD.Pause THEN
		Monitoring.Visu_StepNo := Monitoring.StepNo ;
	ELSIF (Monitoring.StepNo = 0)THEN
		Monitoring.Visu_StepNo := 0 ;
	END_IF
	
	
	rTrigCycleStart(CLK:= CMD.Start);	
	IF rTrigCycleStart.Q AND Status.Running AND Monitoring.StepNo > 0 THEN
		CMD.Start:=	FALSE;		
		fnLogMsg(ADR(LogMsg_0), LOG_ERROR, CONCAT(Parameter.CHName ,' ,Start Command While Cycle Running was ignored, FlowID = %d'),0,0,0);
	END_IF

	
	(*************************** Step By Step *****************************************)
	// Step By Step Logic: If Step By Step bit set:
	//							- We stay at the same step 
	//							- We set the Pause flag
	//							- We whait for Resume bit to set to continue
	(********************************************************************)
	IF CMD.StepByStep AND (CMD.Resume OR ResumeAllTrig.Q) THEN
		CMD.Resume	:=FALSE;
		CMD.Pause	:=FALSE;
	END_IF

	IF (CMD.StepByStep AND LastStepNo <> Monitoring.StepNo)THEN
		CMD.Pause	:=TRUE;
	END_IF

	rTrigCycleDone(CLK := Status.Done);
	IF CMD.StepByStep AND rTrigCycleDone.Q THEN
		CMD.Pause	:=FALSE;
	END_IF

	(*************************** Step Time Out *****************************************)
	// Time Out Logic: If timeout elapsed:
	//							- We set the FAULT flag
	//							- We set the Error_Number and Error_Text
	//							- We set the Pause flag
	(********************************************************************)
	
	//SubStep Stuck
	Status.SubStepStuck :=  (Monitoring.SubStepNo = LastSubStepNo) AND (Status.Running) AND (Monitoring.SubStepNo <> 0);
	LastSubStepNo := Monitoring.SubStepNo;
	
	SubStepTimerTOut.PT := Parameter.TimeOut ;
	SubStepTimerTOut.IN := Status.SubStepStuck
							AND NOT CMD.Pause
							AND NOT CMD.DeactivateStepTimeOut ;
					
	SubStepTimerTOut();
	Monitoring.SubStep_TimeOut := SubStepTimerTOut.ET ;

	//Step Stuck
	Status.CycleStuck:= (LastStepNo = Monitoring.StepNo)
			 AND (Status.Running) 
			 AND Monitoring.SubStepNo = 0 ;
			
	
	StepTimerTOut.PT := Parameter.TimeOut ;
	StepTimerTOut.IN := Status.CycleStuck
							AND NOT CMD.Pause
							AND NOT CMD.StepByStep
							AND NOT CMD.DeactivateStepTimeOut ;					
	StepTimerTOut();

	Monitoring.Step_TimeOut := StepTimerTOut.ET ;
	
	
	IF StepTimerTOut.Q OR SubStepTimerTOut.Q OR SetEvent THEN
		SetEvent := FALSE ;
		Status.Fault:=	TRUE;
		TimeOutFault:=	TRUE;
	END_IF
	
		 
	IF Status.Fault THEN
		CMD.Pause := TRUE;
	END_IF

	// Logging & Event
	IF Triger2.EDGEPOS(Status.Fault) THEN
		IF TimeOutFault THEN
			IF 	Monitoring.Error_Text = Monitoring.StepMessage THEN
				fnLogMsg(ADR(LogMsg_0),
				 LOG_ERROR,
					CONCAT(
						CONCAT(
							CONCAT(Parameter.CHName,', State = %d ,SubState = %d, FlowID = %d,'),
																					Monitoring.Error_Text),
																					' ,Fault - Time Out Elaspsed'),
																						Monitoring.StepNo,
																						Monitoring.SubStepNo,0);
			ELSE
				fnLogMsg(ADR(LogMsg_0),
				 LOG_ERROR,
					CONCAT(
						CONCAT(
							CONCAT(Parameter.CHName,', State = %d ,SubState = %d, FlowID = %d,'),
																					Monitoring.Error_Text),
																					' Fault - By Event'),
																						Monitoring.StepNo,
																						Monitoring.SubStepNo,0);
			END_IF	

		//	IF NOT __ISVALIDREF(rEvent) THEN
		//		//rEvent REF=	ev_PLC_INTERNAL_TIMEOUT;	
		//		Monitoring.ExternalLogText := 'No Link to Event, send default PLC internal Timeout event';
		//		CMD.WriteExternalFaultLogCMD := TRUE;
		//	END_IF
			//fbCHPrgmBasic.mEventThrow(rEvent,ADR(EventHeader),ADR(EventParameters));
				
		ELSE
			
			fnLogMsg(ADR(LogMsg_0),
			 LOG_ERROR,
				CONCAT(
					CONCAT(
						CONCAT(Parameter.CHName,', State = %d ,SubState = %d, FlowID = %d ,'),
																				Monitoring.Error_Text),
																				' Fault - By External Event'),
																					Monitoring.StepNo,
																					Monitoring.SubStepNo,0);
		
			//Event Parames reset
			//memset(ADR(EventParameters),0,SIZEOF(EventParameters)) ;
		END_IF
		
		
	END_IF
	
	IF CMD.WriteExternalFaultLogCMD THEN
		CMD.WriteExternalFaultLogCMD := FALSE ;
		fnLogMsg(ADR(LogMsg_0), LOG_INFO, CONCAT(CONCAT(Parameter.CHName , Monitoring.ExternalLogText), ', ERROR ID = %d, FlowID = %d.'),Monitoring.ExternalLogParam1,0,0);
	END_IF
	
	IF CMD.WriteExternalLogCMD THEN
		CMD.WriteExternalLogCMD := FALSE ;
		//fnLogMsg(ADR(LogMsg_0), Parameter.ExternalLogType, CONCAT(CONCAT(Parameter.CHName,', '), Monitoring.ExternalLogText),0,0,0);
		fnLogMsg(ADR(LogMsg_0), Parameter.ExternalLogType, CONCAT(CONCAT(CONCAT(Parameter.CHName, ', ') , Monitoring.ExternalLogText), ' %d '),Monitoring.ExternalLogParam1,0,0);
	END_IF
	
	
	//StepOneShotTrig	- After Fault Handling
	IF (Monitoring.StepNo <> LastStepNo) THEN
		PrevStepNo := LastStepNo;
		LastStepNo := Monitoring.StepNo ;
		Monitoring.LastStep:= LastStepNo;
		StepOneShotTrig:=	TRUE;
		Monitoring.SubStepNo:=	0;
		//rEvent REF=	ev_PLC_INTERNAL_TIMEOUT;	
	ELSE
		StepOneShotTrig:=	FALSE;
	END_IF
	
	
	
	(*************************** Reset All *****************************************)
	// Reset All: If ResetCycle^ CMD Executed:
	//							- We reset the FAULT flag
	//							- We reset the Error_Number and Error_Text
	//							- We reset the Pause flag
	//							- We reset the Cycle^Stuck flag
	//							- We reset the Running flag
	//							- We reset the Done flag
	//							- We reset the StepNo 
	//							- We reset the StepMessage
	//							- We reset the StepByStep flag
	//							- We reset the NoFaultStep flag
	//							- We reset the ResetCycle^ flag
	//							- We reset the Delay Timer
	//							- We reset the Cycle^TimeOut_Fault flag
	(********************************************************************)	
	

	IF CMD.ResetCycle THEN
//		fnLogMsg(ADR(LogMsg_0), LOG_INFO, CONCAT(CONCAT(Parameter.CHName,', State = %d, FlowID = %d '),'Reset Cycle'),Monitoring.StepNo,pFlowID^,0);
		fnLogMsg(ADR(LogMsg_0), LOG_INFO, CONCAT(CONCAT(Parameter.CHName,', Reset Cycle, '),'State = %d.'),Monitoring.StepNo,0,0);
		Status.Fault 					:= FALSE;
		TimeOutFault					:= FALSE;
		Status.CycleStuck 				:= FALSE;
		CMD.Start 						:= FALSE;
		Status.Running 					:= FALSE;
		Status.Done 					:= FALSE;
		CMD.Pause 						:= FALSE;
		Monitoring.StepNo 				:= 0;
		Monitoring.PrevStepNo 			:= 0;
		Monitoring.SubStepNo 			:= 0;
		Monitoring.StepMessage 			:= '';
		CMD.StepByStep 					:= FALSE;
		CMD.DeactivateStepTimeOut 		:= FALSE;
		CMD.ResetCycle 					:= FALSE;
		Monitoring.Error_Text 			:= '' ;
		Monitoring.External_Error_Text 	:= '' ;
		Monitoring.ExternalLogText		:= '' ;
		Delay.IN 						:= FALSE ;
		Delay();
		Status.CycleTimeOut_Fault 		:= FALSE ;
		LastStepNo 						:= 0 ;
		LastStepMessage 				:= '';			
	END_IF
	
	
	(*************************** Resume the Cycle^ from last step ***************************)
	// Resume Logic: If No Fault and Resume bit set:
	//							- We reset the Cycle^Stuck flag
	//							- We reset the Resume
	//							- We reset the Pause flag
	(********************************************************************)
	IF NOT Status.Fault AND CMD.Resume THEN
		fnLogMsg(ADR(LogMsg_0), LOG_INFO, CONCAT(CONCAT(Parameter.CHName,', Resume, '),'State = %d.'),Monitoring.StepNo,0,0);
//		fnLogMsg(ADR(LogMsg_0), LOG_INFO, CONCAT(CONCAT(Parameter.CHName,', State = %d, FlowID = %d '),'Resume'),Monitoring.StepNo,pFlowID^,0);
		CMD.Pause 			:= FALSE;
		Status.CycleStuck 	:= FALSE;
		CMD.Resume 			:= FALSE;
		StepOneShotTrig		:= TRUE;
	END_IF

	
	(*************************** Auto Errors Reset ***************************)
	// Errors Logic: If No Fault and not Cycle^TimeOut_Fault:
	//							- We reset the Error_Num 
	//							- We reset the Error_Text
	(********************************************************************)
	IF NOT Status.Fault AND NOT Status.CycleTimeOut_Fault THEN
		Monitoring.Error_Text 			:= '' ;
		Monitoring.External_Error_Text 	:= '' ;
	END_IF
	
	
	(*************************** Errors Reset ***************************)
	// Errors Logic: If ResetErr bit set:
	//							- We reset the Error_Num 
	//							- We reset the Error_Text
	//							- We reset the Pause flag
	//							- We reset the Fault flag
	//							- We reset the Cycle^TimeOut_Fault flag
	(********************************************************************)
	//ResetFaultTrig.CLK := CMD.ResetErr ;
	//ResetFaultTrig();
	IF (*ResetFaultTrig.Q*)CMD.ResetErr THEN
		CMD.ResetErr := FALSE ;
		fnLogMsg(ADR(LogMsg_0), LOG_INFO, CONCAT(CONCAT(Parameter.CHName,', Reset Error, '),'State = %d, FlowID = %d.'),Monitoring.StepNo,0,0);
		Monitoring.Error_Text 			:= '' ;
		Monitoring.External_Error_Text 	:= '' ;
		
		Status.Fault 					:= FALSE ;
		TimeOutFault					:= FALSE ;
		Status.CycleTimeOut_Fault 		:= FALSE ;
	END_IF
	
	
	//Cycle^ TIME
	IF CMD.Deacivate_Sequence_Time_Out = FALSE THEN
		(*************************** Monitoring Last Cycle^ Time ***************************)
		// Last Cycle^ Time Logic: If Running flag bit set:
		//						  - We set the LastCycle^Time to Cycle^Time.ET
		(********************************************************************)
		fTrigCycleRunning.CLK			:= Status.Running ;
		fTrigCycleRunning();
		IF fTrigCycleRunning.Q THEN
			Monitoring.LastCycleTIME 	:= CycleTIME.ET;
		END_IF
	
 
		(*************************** Seting the tiem of Cycle^ Time Out ***************************)
		// Cycle^ Time Out Logic: If Cycle^TimeOut > 0:
		//						  - We set the Cycle^Time.PT to Cycle^TimeOut
		(********************************************************************)
		IF TIME_TO_DINT(Parameter.CycleTimeOut) > 0 THEN
			CycleTIME.PT := (Parameter.CycleTimeOut) ;
		ELSE
			CycleTIME.PT := T#30M ;
		END_IF
		
		(*************************** Cycle^ Time set ***************************)
		// Cycle^ Time set Logic: If Running and not Cycle^TimeOut_Fault and not Deacivate_Sequence_Time_Out :
		//						  - We set the Cycle^Time.IN 
		(********************************************************************)
		CycleTIME.IN := Status.Running AND NOT Status.CycleTimeOut_Fault (*AND NOT CMD.Deacivate_Sequence_Time_Out *);
		CycleTIME();
		
		
		(*************************** Cycle^ Time Out ***************************)
		// Cycle^ Time Out Logic: If Cycle^Time.Q bit set:
		//							- We set the Error_Text
		//							- We set the Pause flag
		//							- We set the Cycle^TimeOut_Fault flag
		(********************************************************************)
		IF CycleTIME.Q THEN
			CMD.Pause 					:= TRUE ;
			Status.CycleTimeOut_Fault 	:= TRUE ;
			Monitoring.Error_Text 		:= 'Sequence Time Out' ;
		END_IF
		
		Monitoring.CycleTIME 	:= CycleTIME.ET ;
	END_IF
	

	

	
	//fbCHPrgmBasic();

	//fnLogTransfer FUNCTION call
	fnLogTransfer(ADR(LogMsg_0));
END_METHOD

PROPERTY PUBLIC CHName : STRING
GET
CHName := THIS^.Parameter.CHName ;
END_GET
SET
THIS^.Parameter.CHName := CHName ;
END_SET
END_PROPERTY

PROPERTY PUBLIC CycleTimeOut : TIME
GET
CycleTimeOut := THIS^.Parameter.CycleTimeOut ;
END_GET
SET
THIS^.Parameter.CycleTimeOut := CycleTimeOut ;
END_SET
END_PROPERTY

PROPERTY PUBLIC Deacivate_Sequence_Time_Out : BOOL
GET
Deacivate_Sequence_Time_Out := THIS^.CMD.Deacivate_Sequence_Time_Out ;
END_GET
SET
THIS^.CMD.Deacivate_Sequence_Time_Out := Deacivate_Sequence_Time_Out ;
END_SET
END_PROPERTY

PROPERTY PUBLIC DeactivateStepTimeOut : BOOL
GET
DeactivateStepTimeOut := THIS^.CMD.DeactivateStepTimeOut ;
END_GET
SET
THIS^.CMD.DeactivateStepTimeOut := DeactivateStepTimeOut ;
END_SET
END_PROPERTY

PROPERTY PUBLIC Done : BOOL
GET
Done := THIS^.Status.Done ;
END_GET
END_PROPERTY

PROPERTY PUBLIC Error_Text : STRING
GET
Error_Text := THIS^.Monitoring.Error_Text ;
END_GET
SET // PUBLIC
THIS^.Monitoring.Error_Text := Error_Text;
END_SET
END_PROPERTY

PROPERTY PUBLIC ExternalLogParam1 : DINT
GET
ExternalLogParam1 := THIS^.Monitoring.ExternalLogParam1;
END_GET
SET
THIS^.Monitoring.ExternalLogParam1 := ExternalLogParam1;
END_SET
END_PROPERTY

PROPERTY PUBLIC ExternalLogText : STRING
GET
ExternalLogText := THIS^.Monitoring.ExternalLogText ;
END_GET
SET
THIS^.Monitoring.ExternalLogText := ExternalLogText ;
END_SET
END_PROPERTY

PROPERTY PUBLIC Fault : BOOL
GET
Fault := THIS^.Status.Fault ;
END_GET
SET
THIS^.Status.Fault := Fault ;
END_SET
END_PROPERTY

PROPERTY PUBLIC LogEnable : BOOL
SET
CMD.EnableStateLogging:= LogEnable ;
END_SET
END_PROPERTY

PROPERTY PUBLIC Pause : BOOL
GET

	Pause := THIS^.CMD.Pause ;
END_GET
SET
 
	THIS^.CMD.Pause := Pause ;
END_SET
END_PROPERTY

PROPERTY PUBLIC pLogMsg_0 : POINTER TO LogMsg
GET
pLogMsg_0:= ADR(THIS^.LogMsg_0);
END_GET
END_PROPERTY

PROPERTY PUBLIC PosForLog : USINT
SET
THIS^.Parameter.PosForLog := PosForLog ;
END_SET
END_PROPERTY

PROPERTY PUBLIC PrevStepNo : DINT
GET
PrevStepNo := THIS^.Monitoring.PrevStepNo ;
END_GET
SET
THIS^.Monitoring.PrevStepNo := PrevStepNo;
END_SET
END_PROPERTY

PROPERTY PUBLIC ResetCycle : BOOL
SET

THIS^.CMD.ResetCycle := ResetCycle ;
END_SET
END_PROPERTY

PROPERTY PUBLIC ResetErr : BOOL
SET
THIS^.CMD.ResetErr := ResetErr ;
END_SET
END_PROPERTY

PROPERTY PUBLIC Resume : BOOL
SET
THIS^.CMD.Resume := Resume ;
END_SET
END_PROPERTY

PROPERTY PUBLIC Running : BOOL
GET
Running := This^.Status.Running ;
END_GET
END_PROPERTY

METHOD SetStepNoWithName
VAR_INPUT
	stepNpmber : DINT;
END_VAR
VAR_IN_OUT
	stateNames : ARRAY [*] OF STRING(32); // in only
END_VAR
StepNo										:= stepNpmber;
Parameter.StepMessageIsForNewState	:= TRUE;;
IF (stepNpmber >= LOWER_BOUND(stateNames,1) AND stepNpmber <= UPPER_BOUND(stateNames,1)) THEN
	Monitoring.StepMessage			:= stateNames[stepNpmber];
ELSE
	Monitoring.StepMessage			:= 'NO_Name_Step';
END_IF
END_METHOD

PROPERTY PUBLIC Start : BOOL
GET

Start := THIS^.CMD.Start ;
END_GET
SET

 THIS^.CMD.Start := Start ;
END_SET
END_PROPERTY

PROPERTY PUBLIC StepByStep : BOOL
GET

StepByStep := THIS^.CMD.StepByStep ;
END_GET
SET
THIS^.CMD.StepByStep := StepByStep ;
END_SET
END_PROPERTY

PROPERTY PUBLIC StepMessage : STRING
GET
StepMessage := THIS^.Monitoring.StepMessage ;
END_GET
SET
THIS^.Monitoring.StepMessage := StepMessage ;
END_SET
END_PROPERTY

PROPERTY PUBLIC StepNo : DINT
GET
StepNo := THIS^.Monitoring.StepNo ;
END_GET
SET
THIS^.Monitoring.StepNo := StepNo ;
END_SET
END_PROPERTY

PROPERTY PUBLIC StepStuck : BOOL
GET
StepStuck := THIS^.Status.CycleStuck;
END_GET
END_PROPERTY

PROPERTY SubStepNo : DINT
GET
SubStepNo := THIS^.Monitoring.SubStepNo ;
END_GET
SET
THIS^.Monitoring.SubStepNo := SubStepNo ;
END_SET
END_PROPERTY

PROPERTY PUBLIC SubStepStuck : BOOL
GET
SubStepStuck := THIS^.Status.SubStepStuck;
END_GET
END_PROPERTY

PROPERTY PUBLIC ThreadName : STRING
GET
ThreadName := THIS^.Parameter.ThreadName ;
END_GET
SET
THIS^.Parameter.ThreadName := ThreadName ;
END_SET
END_PROPERTY

PROPERTY PUBLIC TimeOut : TIME
GET
TimeOut := THIS^.Parameter.TimeOut ;
END_GET
SET
THIS^.Parameter.TimeOut := TimeOut ;
END_SET
END_PROPERTY

PROPERTY WriteExternalFaultLog : BOOL
SET
 THIS^.CMD.WriteExternalFaultLogCMD := WriteExternalFaultLog ;
END_SET
END_PROPERTY

PROPERTY WriteExternalLog : BOOL
GET
WriteExternalLog:= THIS^.CMD.WriteExternalLogCMD;
END_GET
SET
 THIS^.CMD.WriteExternalLogCMD := WriteExternalLog ;
END_SET
END_PROPERTY

END_FUNCTION_BLOCK

// ---- POUs/Lib/Logging/logLib/LogMsg.TcPOU
FUNCTION_BLOCK LogMsg
VAR_INPUT
	operationType :OperationTypeEnum ; (*Which operation to do: writing to local array or move from local to global array*)	
	Enable : BOOL;
	ptrEncoderAngle : POINTER TO REAL;
	ptrGlobalArray : POINTER TO LogGlobalArrayObj; (*Address of global array*)
	logData : LogMsgLogData; (*Log data, moved to function block, after using need to be cleared*)	
END_VAR
VAR_OUTPUT
	ErrorID : USINT;	
END_VAR
VAR_STAT
	UseFunctionSuppressBlank : BOOL := TRUE;
END_VAR

VAR

	logLocalArray : LogLocalArrayObj;
	//globalArray : REFERENCE TO LogGlobalArrayObj; (*Pointer of global array structure*)
	tempIndex : UINT;
	//encoderAngle : REFERENCE TO REAL;
	MembersToWrite	: UINT;	
	i 				: UINT;	
	NT_GetTime_0 : NT_GetTime;
	
	FB_FormatString_0:FB_FormatString;
END_VAR


CASE operationType OF
	(* Copy log message to local array *)
	COLLECT2LOCAL:
	
		IF Enable THEN (* Writing to local array only if enabled *)
			IF logLocalArray.pointers.numOfMembers < LOCAL_ARRAY_LENGTH THEN
				(* Copies data to local structure *)
				tempIndex := logLocalArray.pointers.writePointer;
				logLocalArray.array_tc[tempIndex].data := logData;
				logLocalArray.array_tc[tempIndex].TIME_TC := RTC.TimeStamp_GMT;
				//NT_GetTime_0(NETID:= ,START := TRUE,TMOUT:= ,BUSY:=,ERR:=,ERRID:= , TIMESTR=>logLocalArray.array_tc[tempIndex].TIME_TC );
				//NT_GetTime_0(START := FALSE);
				//RTC_gettime(ADR(logLocalArray.array_tc[tempIndex].TIME_TC));
				//encoderAngle ACCESS encoderAngleAddr;
				//Translates from PLC angle (0..360000) to normal angle units (0..720 degrees)
				logLocalArray.array_tc[tempIndex].Angle := REAL_TO_UINT(ptrEncoderAngle^);  //Oren// REAL_TO_UINT(floor_f((ptrEncoderAngle^*2+500)/1000.0));
				logLocalArray.pointers.writePointer := (tempIndex + 1) MOD LOCAL_ARRAY_LENGTH;
				logLocalArray.pointers.numOfMembers := logLocalArray.pointers.numOfMembers + 1;
			ELSE
				ErrorID := 1;
			END_IF;
		END_IF;	
	(* Copy all messages from local array to global array *)
	COPY2GLOBAL:

		//globalArray ACCESS globalArrayAddr;
		(*IF ptrGlobalArray^.SemData.SemID = 0 THEN
			IF globalArray.SemData.SemCreate_0.status = 0 THEN  (* SemCreate successful *)
				globalArray.SemData.SemID := globalArray.SemData.SemCreate_0.ident;  (* copy semaphore-ident the a gobal variable for global use *)
 				SemRelease(globalArray.SemData.SemID);  (* release the allocated semaphore *)
			ELSIF globalArray.SemData.SemCreate_0.status = ERR_FUB_BUSY THEN
				globalArray.SemData.SemCreate_0();
			END_IF	
		END_IF*)   

		IF	// globalArray.SemData.SemID <> 0 AND 
			//AND ptrGlobalArray^.pointers.numOfMembers < GLOBAL_ARRAY_LENGTH THEN
			logLocalArray.pointers.numOfMembers > 0 THEN
			
			IF ptrGlobalArray^.SemData.SemaStat = 0 THEN (*Allocation succesfull *)
				ptrGlobalArray^.SemData.SemaStat :=1;

				MembersToWrite := MIN(logLocalArray.pointers.numOfMembers,
										GLOBAL_ARRAY_LENGTH - ptrGlobalArray^.pointers.numOfMembers);
				MembersToWrite := MIN(MembersToWrite, MAX_MEMBERS_TO_WRITE);
				
				FOR	i := 1 TO MembersToWrite DO							
					ptrGlobalArray^.array_tc[ptrGlobalArray^.pointers.writePointer]	:= logLocalArray.array_tc[logLocalArray.pointers.readPointer];
					ptrGlobalArray^.pointers.writePointer	:= (ptrGlobalArray^.pointers.writePointer + 1)	MOD GLOBAL_ARRAY_LENGTH;
					logLocalArray.pointers.readPointer		:= (logLocalArray.pointers.readPointer + 1)		MOD LOCAL_ARRAY_LENGTH;
				END_FOR;

				logLocalArray.pointers.numOfMembers		:= logLocalArray.pointers.numOfMembers - MembersToWrite;
				ptrGlobalArray^.pointers.numOfMembers	:= ptrGlobalArray^.pointers.numOfMembers + MembersToWrite;
				
				//release semophere
				ptrGlobalArray^.SemData.SemaStat :=0;
				//SemRelease(globalArray.SemData.SemID);
				
			END_IF
		END_IF
END_CASE;

METHOD EnableLogger
VAR_INPUT
	toEnable: BOOL;
END_VAR
Enable := toEnable;
END_METHOD

METHOD FB_init : BOOL
VAR_INPUT
	bInitRetains : BOOL; // if TRUE, the retain variables are initialized (warm start / cold start)
	bInCopyCode : BOOL;  // if TRUE, the instance afterwards gets moved into the copy code (online change)
END_VAR

// beware of overriding initialization has been done by particular user
IF (ptrGlobalArray = 0) THEN
	InitLogger('LogName', 0,0);
	EnableLogger(TRUE);
END_IF
END_METHOD

//
// if globalArrayAddr and/or encoderAngleAddr is set to 0,
// so if InitLogger is called the first time, init it to defaults,
// otherwise, keep values as have been already set. 

METHOD InitLogger : BOOL
VAR_INPUT
	categoryName		: STRING[LOG_MSG_CATEGORY_LENGTH];
	globalArrayAddr		: POINTER TO LogGlobalArrayObj;
	encoderAngleAddr	: POINTER TO REAL;	
END_VAR
	THIS^.logData.category := categoryName;
	
	// if globalArrayAddr and/or encoderAngleAddr is set to 0,
	// so IF InitLogger is called the first time, init it TO defaults,
	// otherwise, keep values as have been already set. 

	IF(globalArrayAddr <> 0) THEN
		THIS^.ptrGlobalArray := globalArrayAddr;
	ELSIF(THIS^.ptrGlobalArray = 0) THEN
		THIS^.ptrGlobalArray := ADR(PcComm.LogGlobalArray);
	END_IF
	
	IF (encoderAngleAddr <> 0)THEN
		THIS^.ptrEncoderAngle := encoderAngleAddr;
	ELSIF (THIS^.ptrEncoderAngle = 0) THEN
		THIS^.ptrEncoderAngle := ADR(CONST_ZERO);
	END_IF

	InitLogger := TRUE;
END_METHOD

METHOD PUBLIC LogMsg : BOOL
VAR_INPUT
		messageLevel : enumLogMessageLevelSeverity;
		textMessage : REFERENCE TO STRING[LOG_MSG_TEXT_LENGTH];
		param1 : DINT;
		param2 : DINT;
		param3 : DINT;
		param4 : DINT;
		param5 : DINT;
		param6 : DINT;
END_VAR
	(* Copying data before putting it into local array *)
	THIS^.logData.levelSeverity := messageLevel;
	THIS^.logData.text := textMessage;
    IF (UseFunctionSuppressBlank=TRUE) THEN
        fnSuppressBlank(ADR(THIS^.logData.text));
    END_IF;
	THIS^.logData.params_tc[0] := param1;
	THIS^.logData.params_tc[1] := param2;
	THIS^.logData.params_tc[2] := param3;
	THIS^.logData.params_tc[3] := param4;
	THIS^.logData.params_tc[4] := param5;
	THIS^.logData.params_tc[5] := param6;
	THIS^.operationType := COLLECT2LOCAL;
	THIS^.logData.noParams := FALSE;	
	THIS^();
	LogMsg := TRUE;
END_METHOD

METHOD LogMsg_v2 : BOOL
VAR_INPUT
		messageLevel : enumLogMessageLevelSeverity;
		textMessage : REFERENCE TO STRING[LOG_MSG_TEXT_LENGTH];
		param1 : T_Arg;
		param2 : T_Arg;
		param3 : T_Arg;
		param4 : T_Arg;
		param5 : T_Arg;
		param6 : T_Arg;
		param7 : T_Arg;
		param8 : T_Arg;
		param9 : T_Arg;
		param10 : T_Arg;		
END_VAR
	(* Copying data before putting it into local array *)
	
	FB_FormatString_0(sFormat := textMessage,arg1 :=param1,arg2 :=param2,arg3 :=param3,arg4 :=param4,arg5 :=param5,arg6 :=param6,arg7 :=param7,arg8 :=param8,arg9 :=param9,arg10 :=param10);
	IF FB_FormatString_0.bError = FALSE THEN
		THIS^.logData.levelSeverity := messageLevel;
		THIS^.logData.text := FB_FormatString_0.sOut;
	ELSE
		THIS^.logData.text := 'Log error, Format text error';
		THIS^.logData.levelSeverity := enumLogMessageLevelSeverity.LOG_ERROR;	
	END_IF	
    IF (UseFunctionSuppressBlank=TRUE) THEN
        fnSuppressBlank(ADR(THIS^.logData.text));
    END_IF;
	THIS^.logData.noParams := TRUE;	

	THIS^.operationType := COLLECT2LOCAL;
	THIS^();
	LogMsg_v2 := TRUE;
END_METHOD

METHOD LogTransfer : BOOL
THIS^.operationType := COPY2GLOBAL;
THIS^();
LogTransfer := TRUE;
END_METHOD

END_FUNCTION_BLOCK

// ---- POUs/Lib/Logging/PLC_ClientComm/UDP_Comm/PcComm/RTC.TcPOU
PROGRAM RTC 
VAR
	FB_LocalSystemTime_0	: FB_LocalSystemTime;
	TimeStamp		: TIMESTRUCT;
		
	TimeStamp_GMT		: TIMESTRUCT;
	
	FB_GetTimeZoneInformation_0 :FB_GetTimeZoneInformation;
	FB_SetTimeZoneInformation_0	:FB_SetTimeZoneInformation;
	ST_TimeZoneInformation:ST_TimeZoneInformation;

	
	Timer :ton;
	FlagGetTimeZone:BOOL;// :=TRUE;
	FlagSetTimeZone:BOOL;// :=TRUE;
	FlagInit	   :BOOL :=TRUE;	
	
	ErrorIDGetTimeZone:UDINT;
	ErrorIDSetTimeZone:UDINT;
	
	FB_TzSpecificLocalTimeToSystemTime:FB_TzSpecificLocalTimeToSystemTime;
//	amsid:T_AmsNetID :='192.168.101.2.1.1' ;
	amsid:T_AmsNetID ;
	
	//IISreset
	NT_StartProcess:NT_StartProcess;
	Flagiisreset:BOOL;
END_VAR

//Timer(IN:=FlagInit,PT:=T#5S,Q=>FlagGetTimeZone);

FB_LocalSystemTime_0(
	sNetID:= '' , 
	bEnable:= TRUE, 
	dwCycle:= , 
	dwOpt:= , 
	tTimeout:= , 
	bValid=> , 
	systemTime=> TimeStamp, 
	tzID=> );

IF FlagInit THEN
	FlagGetTimeZone:=TRUE;
	Flagiisreset:=TRUE;
	FlagInit:=FALSE;
	
END_IF	

	FB_GetTimeZoneInformation_0(bExecute := FlagGetTimeZone,sNetID:=PcTransmit.fbPcTransmit_0.RTC_amsid);
	IF FB_GetTimeZoneInformation_0.bError THEN
		FlagGetTimeZone:=FALSE;
		ErrorIDGetTimeZone:=FB_GetTimeZoneInformation_0.nErrID;
		FB_GetTimeZoneInformation_0(bExecute := FlagGetTimeZone);   		
	ELSIF FB_GetTimeZoneInformation_0.bBusy=FALSE AND FlagGetTimeZone THEN
		ST_TimeZoneInformation:=FB_GetTimeZoneInformation_0.tzInfo;	
		FlagGetTimeZone:=FALSE;
		FlagSetTimeZone:=TRUE;
		FB_GetTimeZoneInformation_0(bExecute := FlagGetTimeZone);	
	END_IF


	FB_SetTimeZoneInformation_0(bExecute:=FlagSetTimeZone, tzInfo:=ST_TimeZoneInformation);
	IF FB_SetTimeZoneInformation_0.bError THEN
		FlagSetTimeZone:=FALSE;
		ErrorIDSetTimeZone:=FB_SetTimeZoneInformation_0.nErrID;
		FB_SetTimeZoneInformation_0(bExecute := FlagSetTimeZone);   		
	ELSIF FB_SetTimeZoneInformation_0.bBusy=FALSE AND FlagSetTimeZone THEN
		FlagSetTimeZone:=FALSE;
		FB_SetTimeZoneInformation_0(bExecute := FlagGetTimeZone);	
	END_IF
	

FB_TzSpecificLocalTimeToSystemTime(in:=TimeStamp,tzInfo:=ST_TimeZoneInformation, out=>TimeStamp_GMT);

(*TEMPH:= DINT_TO_INT(ST_TimeZoneInformation.bias+ST_TimeZoneInformation.daylightBias)/60;

Temp_H:=(WORD_TO_INT(TimeStamp.wHour) +TEMPH)MOD(24) ;
IF Temp_H<0 THEN
	Temp_H:=Temp_H+24;
END_IF

TimeStamp_GMT :=TimeStamp;
TimeStamp_GMT.wHour:= INT_TO_WORD(Temp_H);*)

//IISRESET
IF Flagiisreset THEN
	NT_StartProcess.PATHSTR := 'C:\hp\iisreset.bat';
	NT_StartProcess.DIRNAME := 'C:\hp';
	NT_StartProcess.START :=TRUE;
	NT_StartProcess();
	IF NT_StartProcess.BUSY = FALSE THEN
		Flagiisreset:=FALSE;
		NT_StartProcess.START :=FALSE;
		NT_StartProcess();
	END_IF
END_IF

END_PROGRAM

// ---- POUs/Lib/Logging/PLC_ClientComm/UDP_Comm/PcComm/PcTransmit.TcPOU
PROGRAM PcTransmit
VAR
	fbPcTransmit_0 : fbPcTransmit;
	//fbLogTransmitMQTT : fbLogTransmitMQTT;
	isMqtt:BOOL;
END_VAR



IF isMqtt THEN
	//fbLogTransmitMQTT();
ELSE
	fbPcTransmit_0();
END_IF

END_PROGRAM

// ---- POUs/Lib/Logging/PLC_ClientComm/UDP_Comm/PcComm/fbPcTransmit.TcPOU
FUNCTION_BLOCK fbPcTransmit
VAR_INPUT

END_VAR
VAR_OUTPUT
	RTC_amsid:T_AmsNetID;
END_VAR
VAR
	
	pGlobalArrayMsg : POINTER TO LogArrayStruct; (*Pointer to global array message, which will be written to the file*)	

	Client : UDPClientHandler_typ ; (*Data for Client Task*)	
	PcSendData : ARRAY[0..UDP_MESSAGE_MAX_LENGTH] OF USINT;
	IgnorePrintDebugMsgsThreshold : UINT;
	ResumePrintDebugMsgsThreshold : UINT;
	IgnorePrintInfoMsgsThreshold : UINT;
	ResumePrintInfoMsgsThreshold : UINT;

	IgnorePrintDebugMsgsFlag : BOOL := FALSE;
	IgnorePrintInfoMsgsFlag : BOOL := FALSE;	
	NumOfRemovedMessages : UINT := 0;	
	logMessagesCount : UINT := 0;
	tempLogMsgCounter : USINT := 0;	
	PcSendDataPtr	: POINTER TO USINT;
	PcSendPackageLenght : UINT;

	intPosition : INT := 0;
	uintPosition : INT := 0;
	hexPosition : INT := 0;	
	pTheFotnat : POINTER TO STRING;
	
	textString : STRING[LOG_MSG_TEXT_LENGTH] := '';	
	paramsCounter : USINT := 0;
	strConverted : STRING[12] := '';
	
	FB_FormatString_0 : FB_FormatString;
	textStringLength : UINT := 0;	
	PcSendDataLenght : USINT := 0;	
	
	LogMsgTime : UDINT := 0;
	SemTakeStatus : UINT;	
	
	//Ftrig1 : F_TRIG;
	//Ftrig2 : F_TRIG;
	Trig1 : Trigger;
	Trig2 : Trigger;
	Trig3 : Trigger;
	Trig4 : Trigger;
	TimerDelayStart : TON ;
	First_Cycle:BOOL;
	
	FaultState:INT;
	FaultTimer:TON;	
	InitDone:BOOL;
END_VAR

VAR CONSTANT
	UDP_PLC_CLIENT_ID : USINT := 91;
	UDP_SERVER_PORT_NUMBER : UINT := 14999;
	UDP_SERVER_ADDRESS : STRING[20] := '192.168.101.15';//'15.17.216.69';//'127.0.0.1';//'192.168.101.15';	
	UDP_SIM_SERVER_ADDRESS: STRING[20] := '127.0.0.1';
	UDP_CLIENT_MAGIC_WORD : UINT := 16#5A5A;
	UDP_MESSAGE_MAX_LENGTH : UDINT := 1400;
	UDP_MAX_NUM_OF_CONT_MSGS : UINT := 5;	
	IGNORED_MSGS_THRESHOLD : UINT := 30;	
	INT_MASK : STRING[2] := '%d';
	UINT_MASK : STRING[2] := '%u';
	HEX_MASK : STRING[2] := '%x';	
	UDP_MESSAGE_HEADER_LENGTH : USINT := 26; (*UDP message header*)	
END_VAR

IF NOT InitDone THEN
	InitDone:=	Meth_PLC_Init();
ELSE
		FaultRecover();
		IF Client.UdpSend_0.bBusy  (*OR Client.UdpSend_0.bExecute = TRUE *) THEN
			 Client.UdpSend_0();
		END_IF	
		IF Trig2.EDGENEG(Client.UdpSend_0.bBusy) OR(NOT(Client.UdpSend_0.bBusy) AND Client.UdpSend_0.bExecute) THEN  
			 Client.UdpSend_0(bExecute := FALSE );
		END_IF			
		IF LogGlobalArray.pointers.numOfMembers > 0 AND Client.UdpSend_0.bBusy = FALSE THEN
			//Client.UdpSend_0(bExecute := FALSE );	(* Call the Function*)
			(* Check if ignore sending INFO and/or DEBUG messages *)
			IF LogGlobalArray.pointers.numOfMembers > IgnorePrintDebugMsgsThreshold THEN
				IgnorePrintDebugMsgsFlag := TRUE;
			ELSIF LogGlobalArray.pointers.numOfMembers < ResumePrintDebugMsgsThreshold THEN
				IgnorePrintDebugMsgsFlag := FALSE;
			END_IF
			
			IF LogGlobalArray.pointers.numOfMembers > IgnorePrintInfoMsgsThreshold THEN
				IgnorePrintInfoMsgsFlag := TRUE;
			ELSIF LogGlobalArray.pointers.numOfMembers < ResumePrintInfoMsgsThreshold THEN
				IgnorePrintInfoMsgsFlag := FALSE;
			END_IF
			
			NumOfRemovedMessages := 0;
			logMessagesCount := MIN(UDP_MAX_NUM_OF_CONT_MSGS, LogGlobalArray.pointers.numOfMembers);
			tempLogMsgCounter := UINT_TO_USINT(logMessagesCount);
			(* Pointers to the start of data structure *)
			PcSendDataPtr := ADR(PcSendData);
			(* Clears send data array *)
			memset(PcSendDataPtr,0,UDP_MESSAGE_MAX_LENGTH);
			(* Putting magic word and number of continuous messages *)
			putUint(UDP_CLIENT_MAGIC_WORD, PcSendDataPtr);
			putUsint(tempLogMsgCounter, PcSendDataPtr);
			PcSendPackageLenght	 := 4;
			WHILE tempLogMsgCounter > 0 AND LogGlobalArray.pointers.numOfMembers > 0 DO
	
				(* Takes message from global array *)
				//pGlobalArrayMsg ACCESS ADR(LogGlobalArray.array[LogGlobalArray.pointers.readPointer]);
				
				pGlobalArrayMsg := ADR(LogGlobalArray.ARRAY_TC[LogGlobalArray.pointers.readPointer]);
				IF ((IgnorePrintDebugMsgsFlag AND pGlobalArrayMsg^.data.levelSeverity = LOG_DEBUG) OR
					(IgnorePrintInfoMsgsFlag AND pGlobalArrayMsg^.data.levelSeverity = LOG_INFO)) AND (NumOfRemovedMessages < IGNORED_MSGS_THRESHOLD) THEN
					(* Need to ignore message *)
					NumOfRemovedMessages := NumOfRemovedMessages +1;
				ELSE
					(* Converts message to string format, the result will be in textString variable *)
					ActionPrintf();
					(* Calculating and adding message length into data *)
					textStringLength := strlen(ADR(textString));
					PcSendDataLenght := UDP_MESSAGE_HEADER_LENGTH + UINT_TO_USINT(textStringLength);
					(* Put message data length*)
					putUsint(PcSendDataLenght, PcSendDataPtr);	
					PcSendPackageLenght := PcSendPackageLenght + PcSendDataLenght;
					(* Adding sequential number internal *)
					putUint(Client.seq_number, PcSendDataPtr);
					Client.seq_number := Client.seq_number + 1;
					(* Adding client ID - constant *)
					putUint(Client.clientId, PcSendDataPtr);
					(* Adding timeStamp (from midnight) from received structure *)
					LogMsgTime := ((pGlobalArrayMsg^.TIME_TC.wHour * 60 + pGlobalArrayMsg^.TIME_TC.wMinute) *60 + pGlobalArrayMsg^.TIME_TC.wSecond)*1000 + pGlobalArrayMsg^.TIME_TC.wMilliseconds;
					putUdint(LogMsgTime,PcSendDataPtr);
					(* Adding encoder angle from received structure*)
					putUint(pGlobalArrayMsg^.Angle,PcSendDataPtr);
					(*Adding sthread name (10 characters) from received structure *)
					putString(ADR(pGlobalArrayMsg^.data.category), LOG_MSG_CATEGORY_LENGTH, PcSendDataPtr);
					(* Adding levelID from received structure *)
					putUsint( DINT_TO_USINT(pGlobalArrayMsg^.data.levelSeverity), PcSendDataPtr);
					(* Addding categoryID - currently not in use *)
					putUdint(0,PcSendDataPtr);
					(* Additng string from textString *)
					putString(ADR(textString), textStringLength, PcSendDataPtr);
					tempLogMsgCounter := tempLogMsgCounter - 1;
				END_IF
				
				LogGlobalArray.pointers.readPointer := (LogGlobalArray.pointers.readPointer + 1) MOD GLOBAL_ARRAY_LENGTH;
				LogGlobalArray.pointers.numOfMembers := LogGlobalArray.pointers.numOfMembers - 1;
			END_WHILE;

			Client.UdpSend_0.cbLen := PcSendPackageLenght;	(* Lenght of data to send *)
			Client.UdpSend_0(bExecute := TRUE );	(* Call the Function*)

			(* For possibility to more effective copies in global array *)
			IF LogGlobalArray.pointers.numOfMembers = 0 AND (LogGlobalArray.pointers.readPointer <> 0 OR LogGlobalArray.pointers.writePointer <> 0) THEN
			    SemTakeStatus := LogGlobalArray.SemData.SemaStat;//  SemAcquire(globalArray.SemData.SemID);
				//SemTakeStatus := SemAcquire(LogGlobalArray.SemData.SemID);
				IF SemTakeStatus = 0 THEN (*Allocation succesfull *)
					LogGlobalArray.SemData.SemaStat :=1;
					IF LogGlobalArray.pointers.numOfMembers = 0 THEN
						LogGlobalArray.pointers.readPointer := 0;
						LogGlobalArray.pointers.writePointer := 0;
					END_IF
					 LogGlobalArray.SemData.SemaStat :=0;
					//SemRelease(LogGlobalArray.SemData.SemID);
				END_IF
			END_IF
		END_IF		
END_IF

ACTION ActionPrintf:
	//textString:='';
	FB_FormatString_0(sFormat := pGlobalArrayMsg^.data.text,
						arg1 := F_DINT( pGlobalArrayMsg^.data.params_tc[0]),
						arg2 := F_DINT( pGlobalArrayMsg^.data.params_tc[1]),
						arg3 := F_DINT( pGlobalArrayMsg^.data.params_tc[2]),
						arg4 := F_DINT( pGlobalArrayMsg^.data.params_tc[3]),
						arg5 := F_DINT( pGlobalArrayMsg^.data.params_tc[4]),
						arg6 := F_DINT( pGlobalArrayMsg^.data.params_tc[5]),
						sOut => textString);
	RETURN;

	strcpy(ADR(textString), ADR(pGlobalArrayMsg^.data.text));
	intPosition := FIND(textString, INT_MASK);
	uintPosition := FIND(textString, UINT_MASK);
	hexPosition := FIND(textString, HEX_MASK);
	paramsCounter := 0;
	WHILE ((intPosition + uintPosition + hexPosition) > 0) AND (paramsCounter <= MAX_COUNT_LOG_PARAM) DO
		IF (intPosition > 0 AND intPosition < uintPosition) THEN
			pTheFotnat := ADR(INT_MASK);
		ELSE	
			pTheFotnat := ADR(UINT_MASK);
			intPosition := uintPosition;
		END_IF
		IF ((hexPosition > 0) AND (intPosition = 0 OR hexPosition < intPosition)) THEN
			textString := DELETE(textString, LEN(HEX_MASK), hexPosition);
			itoax(TO_UDINT(pGlobalArrayMsg^.data.params_tc[paramsCounter]), ADR(strConverted));
			textString := INSERT(textString, strConverted, (hexPosition-1));
		ELSE	
			textString := DELETE(textString, LEN(pTheFotnat^), intPosition);
			FB_FormatString_0(sFormat := pTheFotnat^,arg1 := F_DINT( pGlobalArrayMsg^.data.params_tc[paramsCounter]), sOut => strConverted  );
			//itoa(pGlobalArrayMsg^.data.params_tc[paramsCounter], ADR(strConverted));
			textString := INSERT(textString, strConverted, (intPosition-1));
		END_IF
		paramsCounter := paramsCounter + 1;
		intPosition := FIND(textString, INT_MASK);
		uintPosition := FIND(textString, UINT_MASK);
		hexPosition := FIND(textString, HEX_MASK);
	END_WHILE;
END_ACTION

ACTION FaultRecover:

IF Trig4.EDGEPOS(Client.UdpSend_0.bError) THEN
	FaultState := 10;
END_IF

CASE FaultState OF
 
	
	10: 
		client.SocketCloseAll_0.bExecute:=TRUE;
		Client.status.opened := FALSE; 
		FaultTimer(in:=TRUE,PT:=T#1S);
		IF FaultTimer.Q THEN
			FaultTimer(in:=FALSE,PT:=T#1S);
			FaultState:=20;
		END_IF	
		
	20:
		client.SocketCloseAll_0.bExecute:=FALSE;
		FaultTimer(in:=TRUE,PT:=T#1S);
		IF FaultTimer.Q THEN
			FaultTimer(in:=FALSE,PT:=T#1S);
			FaultState:=30;
		END_IF			
		
	30:
		Client.UdpOpen_0.bExecute 		:= TRUE;
		FaultState:=0;
			
END_CASE

client.SocketCloseAll_0();
END_ACTION

METHOD Meth_PLC_Init : BOOL
VAR_INPUT
END_VAR
VAR_INST
	
	State:	INT;	

END_VAR

CASE State OF  
	0:
		Meth_PLC_Init:=	FALSE;	
		Client.clientId := UDP_PLC_CLIENT_ID; 
		
		Client.UdpOpen_0.nLocalPort 	:= 0;//0;//UDP_SERVER_PORT_NUMBER;	(* Port to listen*)
		Client.UdpOpen_0.tTimeout	    := T#3S;

		Client.Udp_GetLocalAmsNetId(bExecute := TRUE);
		IF Client.Udp_GetLocalAmsNetId.AddrBytes[0] <> 0 THEN
			Client.UdpOpen_0.sSrvNetId 		:= Client.Udp_GetLocalAmsNetId.AddrString;	(* If empty string=>server runs on local system*)
			IF strcmp(ADR(Client.Udp_GetLocalAmsNetId.AddrString), ADR('192.168.101.10.1.1')) = 0 THEN
			//	Client.UdpOpen_0.sSrvNetId 		:= '192.168.101.10.1.1';//'';	(* If empty string=>server runs on local system*)
				Client.UdpOpen_0.sLocalHost 	:= '192.168.101.10';//'';	(* Local address*)
			ELSIF strcmp(ADR(Client.Udp_GetLocalAmsNetId.AddrString), ADR('192.168.102.10.1.1')) = 0 THEN
			//	Client.UdpOpen_0.sSrvNetId 		:= '192.168.102.10.1.1';//'';	(* If empty string=>server runs on local system*)
				Client.UdpOpen_0.sLocalHost 	:= '192.168.102.10';//'';	(* Local address*)
			ELSE
				Client.UdpOpen_0.sSrvNetId 		:= '';	(* If empty string=>server runs on local system*)
				Client.UdpOpen_0.sLocalHost 	:= '';	(* Local address*)			
			END_IF
			TimerDelayStart(in:=TRUE,pt:=T#5S);
		END_IF
		IF Client.status.opened = FALSE THEN
			IF Trig3.EDGEPOS(TimerDelayStart.Q)THEN
				TimerDelayStart(in:=FALSE,pt:=T#5S);
				Client.UdpOpen_0(bExecute := TRUE);	(* Call the Function*)
//			IF (NOT Client.UdpOpen_0.bError) THEN
				IF Trig1.EDGENEG(Client.UdpOpen_0.bBusy) THEN  (* UdpOpen successful*)
					Client.status.opened := TRUE;
					Client.UdpSend_0.hSocket := Client.UdpOpen_0.hSocket;
					IF Client.Udp_GetLocalAmsNetId.AddrBytes[0] <> 0 THEN
						IF strcmp(ADR(Client.Udp_GetLocalAmsNetId.AddrString), ADR('192.168.101.10.1.1')) = 0 THEN
							Client.UdpSend_0.sRemoteHost := '192.168.101.2';//UDP_SERVER_ADDRESS;			
							RTC_amsid := 	'192.168.101.2.1.1';
						ELSIF strcmp(ADR(Client.Udp_GetLocalAmsNetId.AddrString), ADR('192.168.102.10.1.1')) = 0 THEN
							Client.UdpSend_0.sRemoteHost := '192.168.102.2';//UDP_SERVER_ADDRESS;			
							RTC_amsid := 	'192.168.102.2.1.1';
						ELSE
							Client.UdpSend_0.sRemoteHost := Client.UdpOpen_0.hSocket.localAddr.sAddr;
						END_IF
					END_IF
					Client.UdpSend_0.sSrvNetId	 := '';	//If empty string=>server runs on local system
					Client.UdpSend_0.nRemotePort := UDP_SERVER_PORT_NUMBER;		
					Client.UdpSend_0.pSrc		 := ADR(PcSendData);	(* Which data to send *)
					//Client.UdpSend_0.tTimeout := ;
					
					// Thresholds for ignore/resume printing messages
					IgnorePrintDebugMsgsThreshold		:= REAL_TO_UINT(GLOBAL_ARRAY_LENGTH * 0.8);
					ResumePrintDebugMsgsThreshold		:= REAL_TO_UINT(GLOBAL_ARRAY_LENGTH * 0.7);
					IgnorePrintInfoMsgsThreshold		:= REAL_TO_UINT(GLOBAL_ARRAY_LENGTH * 0.6);
					ResumePrintInfoMsgsThreshold		:= REAL_TO_UINT(GLOBAL_ARRAY_LENGTH * 0.5);
					State:=	State + 1;
				//	Client.UdpSend_0.bExecute := TRUE;
				END_IF
			END_IF	
//			END_IF
		END_IF

	1:
		Meth_PLC_Init:=	TRUE;
END_CASE
END_METHOD

END_FUNCTION_BLOCK

// ---- POUs/Lib/Logging/PackData/putUint.TcPOU
FUNCTION putUint : BOOL
	VAR_INPUT
		uintVar : UINT;
	END_VAR
	VAR_IN_OUT
		bufferRef : POINTER TO USINT;
	END_VAR

memcpy(bufferRef, ADR(uintVar), SIZEOF(UINT));
bufferRef := bufferRef + SIZEOF(UINT);
putUint := TRUE;

END_FUNCTION

// ---- POUs/Lib/Logging/PackData/putUsint.TcPOU
FUNCTION putUsint : BOOL
	VAR_INPUT
		usintVar : USINT;
	END_VAR
	VAR_IN_OUT
		bufferRef : POINTER TO USINT;
	END_VAR

	memcpy(bufferRef, ADR(usintVar), SIZEOF(USINT));
	bufferRef := bufferRef + SIZEOF(USINT);
	putUsint := TRUE;

END_FUNCTION

// ---- POUs/Lib/Logging/HpString/strlen.TcPOU
FUNCTION strlen : UINT
VAR_INPUT
	pStr	: POINTER TO STRING;
END_VAR
VAR
	tmpStrLen	: UINT;
	pArr		: POINTER TO BYTE;
END_VAR

(********************************************************************
 * COPYRIGHT -- Hewlett-Packard Company
 ********************************************************************
 * Program: logLib
 * File: logLib.st
 * Author: 
 * Created: Feb 20, 2017
 ********************************************************************
 * Implementation of program logLib
 ********************************************************************) 

tmpStrLen	:= 0;
pArr		:= pStr;
WHILE pArr^ <> 0 DO
	tmpStrLen	:= tmpStrLen + 1;
	pArr	:= pArr + 1;
END_WHILE
strlen	:= tmpStrLen;
RETURN;

END_FUNCTION

// ---- POUs/Lib/Logging/PackData/putUdint.TcPOU
FUNCTION putUdint : BOOL
	VAR_INPUT
		udintVar : UDINT;
	END_VAR
	VAR_IN_OUT
		bufferRef : POINTER TO USINT;
	END_VAR

	memcpy(bufferRef, ADR(udintVar), SIZEOF(UDINT));
	bufferRef := bufferRef + SIZEOF(UDINT);
	putUdint := TRUE;

END_FUNCTION

// ---- POUs/Lib/Logging/PackData/putString.TcPOU
FUNCTION putString : bool
	VAR_INPUT
		stringPtr : POINTER TO STRING;
		stringLength : UINT;
	END_VAR
	VAR_IN_OUT
		bufferRef : POINTER TO USINT;
	END_VAR

	memcpy(bufferRef, stringPtr, stringLength);
	bufferRef := bufferRef + stringLength;
	putString := TRUE;

END_FUNCTION

// ---- POUs/Lib/Logging/HpString/strcpy.TcPOU
FUNCTION strcpy : UDINT
VAR_INPUT
	pDst : POINTER TO STRING;
	pSrc : POINTER TO STRING;
END_VAR
VAR
	pArr		: POINTER TO BYTE;
	pArrDst		: POINTER TO BYTE;
END_VAR

pArr		:= pSrc;
pArrDst		:= pDst;
WHILE (pArr^ <> 0)  DO
	pArrDst^ := pArr^;

	pArr := pArr+1;
	pArrDst := pArrDst+1;

END_WHILE
pArrDst^ := pArr^;

END_FUNCTION

// ---- POUs/Lib/Logging/HpString/itoax.TcPOU
FUNCTION itoax : UINT  (*Create a string with hex digits of value*)
VAR_INPUT
		Value : UDINT; (*Number for conversion to string*)
		pString : POINTER TO STRING; (*Pointer to destination string*)	
END_VAR
VAR
	hexString : ARRAY[0..5] OF USINT;
	Digit : UDINT;
	byteDigit : POINTER TO USINT;
	idx : USINT;	
END_VAR

	//byteDigit ACCESS ADR(Digit);
	byteDigit := ADR(Digit);
	FOR idx := 0 TO 3 DO
		Digit := Value AND 16#000F;
		IF Digit < 10 THEN 						// 0-9
			hexString[3-idx] := byteDigit^ + 48; // digit+'0'  
		ELSE									// A-F
			hexString[3-idx] := byteDigit^ + 55; // digit+'A'-10
		END_IF
		Value := SHR(Value,4);
	END_FOR
	hexString[4] := 72; 						// 'H' suffix
	hexString[5] := 0;							// Null terminator
	memcpy(pString,ADR(hexString[0]),SIZEOF(hexString));
	itoax := SIZEOF(hexString);

END_FUNCTION

// ---- POUs/Lib/Logging/HpString/strcmp.TcPOU
FUNCTION strcmp : DINT
VAR_INPUT
	pStr1 : POINTER TO STRING;
	pStr2 : POINTER TO STRING;
END_VAR
VAR
	pArr1	: POINTER TO BYTE;
	pArr2	: POINTER TO BYTE;
	dif		: DINT;
END_VAR


pArr1		:= pStr1;
pArr2		:= pStr2;
WHILE (pArr1^ <> 0 OR pArr2^ <> 0) AND_THEN dif = 0 DO	
	dif	:= pArr1^ - pArr2^;
	pArr1 := pArr1+1;
	pArr2 := pArr2+1;
END_WHILE

strcmp := dif;

END_FUNCTION

// ---- POUs/Lib/Logging/logLib/fnSuppressBlank.TcPOU
FUNCTION fnSuppressBlank : BOOL
VAR_INPUT
	pStr		: POINTER TO STRING;
	//stringAdr : UDINT := 0;		
END_VAR

VAR
		//Str : REFERENCE TO STRING[256];
		position : UINT := 0;
		StringLen : UINT := 0;
		SpacesNum : UINT := 0; (*number of spacess*)
		PrevIsLetter : BOOL := FALSE; (* it is true, if previous character is letter *)
		WordsNum : UINT := 0; (*number of words*)
		nxt_adr : UDINT := 0;
		LettersNumber : UINT := 0; (*number of letters*)
		WordLen : UINT := 0;	
END_VAR

   // Str ACCESS stringAdr;//reference to string
    StringLen:=strlen(pStr);
    nxt_adr :=memmove(pStr+StringLen,ADR(' '),  1); // put the space to last place, for optimization of the algorithm 
    FOR position:=0 TO StringLen DO
        IF (memcmp(pStr+position,ADR(' '),1)=0) OR (memcmp(pStr+position,ADR(' '),1)=0) THEN  //it is space
            SpacesNum:=SpacesNum+1;
            IF (PrevIsLetter=TRUE) THEN
                IF (SpacesNum>WordsNum) THEN //last word not in his place
                    nxt_adr :=memmove(pStr+LettersNumber+WordsNum, pStr+position-WordLen,  WordLen+1); // Move the word to its place
                END_IF;
                WordsNum:=WordsNum+1;
                LettersNumber:=LettersNumber+WordLen;
                WordLen:=0;
                PrevIsLetter:=FALSE;
            END_IF;
        ELSE
            PrevIsLetter:=TRUE;
            WordLen:=WordLen+1;
        END_IF;
    END_FOR;
    nxt_adr :=memmove(pStr+LettersNumber+WordsNum-1,ADR(''),  1); // put the end of line to its place
    IF (LettersNumber+WordsNum>StringLen) OR (StringLen=0) THEN
        fnSuppressBlank:=FALSE;//the function did not change the string
    ELSE 
        fnSuppressBlank:=TRUE;//the function changed the string
    END_IF;

END_FUNCTION

// ---- POUs/Lib/Logging/logLib/fnLogMsgInit.TcPOU
FUNCTION fnLogMsgInit : BOOL
VAR_INPUT
		//logMsgPtr : REFERENCE TO LogMsg;
		logMsgPtr 		 : POINTER TO LogMsg;
		category  		 : STRING[LOG_MSG_CATEGORY_LENGTH];
		globalArrayAddr  : POINTER TO LogGlobalArrayObj;
		encoderAngleAddr : POINTER TO REAL;	
END_VAR
VAR
	
END_VAR

	fnLogMsgInit := logMsgPtr^.InitLogger(category, globalArrayAddr, encoderAngleAddr);

END_FUNCTION

// ---- POUs/Lib/Logging/logLib/fnLogMsg.TcPOU
FUNCTION fnLogMsg : BOOL
VAR_INPUT
		logMsgPtr : POINTER TO LogMsg;
		messageLevel : enumLogMessageLevelSeverity;
		textMessage : STRING[LOG_MSG_TEXT_LENGTH];
		param1 : DINT;
		param2 : DINT;
		param3 : DINT;
END_VAR

fnLogMsg := logMsgPtr^.LogMsg(messageLevel, textMessage, param1, param2, param3, 0, 0, 0);

END_FUNCTION

// ---- POUs/Lib/Logging/logLib/fnLogTransfer.TcPOU
FUNCTION fnLogTransfer : BOOL
VAR_INPUT
	logMsgPtr : POINTER TO LogMsg;
END_VAR
VAR
END_VAR


fnLogTransfer := logMsgPtr^.LogTransfer();

END_FUNCTION

// ---- POUs/App/FB_RW_Ctrl.TcPOU
FUNCTION_BLOCK FB_RW_Ctrl EXTENDS CycleHandleFB
VAR_INPUT
	Ctrl_ref:			REFERENCE TO Ctrl_Typ;
END_VAR
VAR_OUTPUT
END_VAR
VAR
	MethInitDone:		BOOL;
END_VAR

VAR CONSTANT
// States are global
		
	RW_INIT:						INT:=0;
	RW_RUN:						INT:=10;
	RW_DONE:			INT:=100;
END_VAR

	IF NOT MethInitDone THEN
		MethInitDone	:= Meth_Init();
	END_IF
	
	IF  THIS^.CMD.Pause = FALSE THEN
		
		//-----------------------------
		//State Machine
		//-----------------------------
		CASE THIS^.StepNo OF
			RW_INIT:
				IF THIS^.StepOneShotTrig THEN
					THIS^.Monitoring.StepMessage	:= 'Init: Start.';
					THIS^.Delay(IN:=FALSE);
				ELSIF Meth_Enable(TRUE) THEN
					THIS^.StepNo	:= 	RW_RUN;
				END_IF	
			
			RW_RUN:
				IF THIS^.StepOneShotTrig THEN
					THIS^.Monitoring.StepMessage	:= 'RW Run.';
					THIS^.Delay(IN:=FALSE);
					Meth_Run_OpenLoop(FALSE);
				ELSIF Meth_Run_OpenLoop(TRUE) THEN
					THIS^.StepNo	:= 	RW_DONE;
				END_IF					
				

			RW_DONE:
				IF THIS^.StepOneShotTrig THEN
					THIS^.Monitoring.StepMessage	:= 'RW cycle Done';
				ELSIF Meth_Done(TRUE) THEN
					THIS^.StepNo	:= 	RW_INIT;
				END_IF		
	
		END_CASE
	
	ELSE
		THIS^.Monitoring.StepMessage:= 'Pause';
		
		IF THIS^.Status.Fault = TRUE THEN
		//IF Meth_EmStop(TRUE) THEN
				THIS^.CMD.ResetCycle	:= TRUE;		// Reset the all state machine to start point
		//END_IF
			
		END_IF
		
	END_IF
	
	THIS^.Delay();
	THIS^.CH_Logic();
	
	// Reset Meth_EmStop when at Init State
	IF THIS^.Pause = FALSE THEN
		//Meth_EmStop(FALSE);
	END_IF

METHOD PRIVATE Meth_Done : BOOL
VAR_INPUT
	Execute: 	BOOL;
END_VAR


	//THIS^.Monitoring.StepMessage			:= 'Press 1 engage';
	//THIS^.Monitoring.Error_Text				:= 'Press 1 engage Fail';
	//THIS^.CMD.Deacivate_Sequence_Time_Out	:= TRUE;	// Disable time out to the all sequence
	//THIS^.CMD.DeactivateStepTimeOut			:= TRUE;	// Disable time out to the actual step
	//THIS^.Parameter.TimeOut					:= T#5S;

	THIS^.Status.Done		:= TRUE;
	THIS^.Status.Running	:= FALSE;									
	Meth_Done	:= TRUE;
END_METHOD

METHOD PRIVATE Meth_Enable : BOOL
VAR_INPUT
	Execute: 	BOOL;
END_VAR


IF THIS^.CMD.Start THEN
	
	THIS^.Monitoring.StepMessage			:= 'Start';
	THIS^.Monitoring.Error_Text				:= 'Start Fail';
	THIS^.CMD.Deacivate_Sequence_Time_Out	:= TRUE;	// Disable time out to the all sequence
	THIS^.CMD.DeactivateStepTimeOut			:= TRUE;	// Disable time out to the actual step
	THIS^.Parameter.TimeOut					:= T#0.5S;

	THIS^.CMD.Start			:= FALSE;
	THIS^.Status.Done		:= FALSE;
	THIS^.Status.Running	:= TRUE;
	
	// Reset Commands and Statuses												
	
	Meth_Enable	:= TRUE;
END_IF
END_METHOD

METHOD Meth_Init :BOOL
VAR_INPUT
END_VAR
//resets
Ctrl_ref.IO.EncoderRW.Ctrl.SetCounterCmd:=FALSE;
RwInverter.ctrl.Start:=FALSE;
RwInverter.ctrl.SetVelocity:=0;

Meth_Init:=TRUE;
END_METHOD

METHOD Meth_Rest_IO 
VAR_INPUT
	
END_VAR

RwInverter.ctrl.Start := FALSE;
RwInverter.ctrl.SetVelocity := 0;
END_METHOD

METHOD Meth_Run_OpenLoop : BOOL
VAR_INPUT
	Excute:BOOL;
END_VAR

IF Excute = FALSE THEN
	THIS^.SubStepNo :=0;
ELSIF Excute AND_THEN THIS^.SubStepNo = 0 THEN
	THIS^.SubStepNo :=10;
END_IF


CASE THIS^.SubStepNo OF
	
	0://Wait
		THIS^.Monitoring.SubStepMessage	:= 'Wait';
		Ctrl_ref.IO.EncoderRW.Ctrl.SetCounterCmd:=FALSE;
		
	
	10://Set counter	
		THIS^.Monitoring.SubStepMessage	:= 'Set counter';
		Ctrl_ref.IO.EncoderRW.Ctrl.SetCounterValue:=0;	
		Ctrl_ref.IO.EncoderRW.Ctrl.SetCounterCmd:=TRUE;	
		IF Ctrl_ref.IO.EncoderRW.Status.SetCounterDone
		OR Ctrl_ref.Simulation 	 THEN
			Ctrl_ref.IO.EncoderRW.Ctrl.SetCounterCmd:=FALSE;
			THIS^.SubStepNo				:=20;
		END_IF	
	
	20: //Start motor
		THIS^.Monitoring.SubStepMessage	:= 'Start Motor';
		RwInverter.ctrl.Start:=TRUE;
		RwInverter.ctrl.SetVelocity:= Ctrl_ref.Parameters.MotorVelocity;	
		THIS^.SubStepNo				:=30;
		
	30://Wait position
		THIS^.Monitoring.SubStepMessage	:= 'Wait position';
		IF Ctrl_ref.IO.EncoderRW.Status.CounterValue >= Ctrl_ref.Parameters.DistanceToMove
		OR Ctrl_ref.Simulation THEN
			RwInverter.ctrl.Start:=FALSE;
			RwInverter.ctrl.SetVelocity:= 0;
			Meth_Run_OpenLoop:=TRUE;
		END_IF
END_CASE
END_METHOD

END_FUNCTION_BLOCK

// ---- POUs/App/FB_Machine_Run.TcPOU
FUNCTION_BLOCK FB_Machine_Run EXTENDS CycleHandleFB
VAR_INPUT
	Ctrl_ref:					REFERENCE TO Ctrl_Typ;
	 FB_RW_Ctrl_ref:			REFERENCE TO FB_RW_Ctrl;
END_VAR
VAR_OUTPUT
END_VAR
VAR
	MethInitDone:		BOOL;
	FB_HeaterProtection:FB_HeaterProtection;
END_VAR
VAR CONSTANT

// States are global
(*		
	MACHINE_RUN_INIT:						INT:=0;
	MACHINE_COLD_CUT_VALVE_OPEN:			INT:=10;
	MACHINE_WELD_VALVE_OPEN:				INT:=20;	
	MACHINE_HEATER_ON:						INT:=30;	
	MACHINE_HEATER_OFF:						INT:=40;
	MACHINE_VALVE_CLOSE:					INT:=50;	
	MACHINE_DONE:							INT:=100;	

*)

END_VAR

	IF NOT MethInitDone THEN
		MethInitDone	:= Meth_Init();
	END_IF
	
	
	IF  THIS^.CMD.Pause = FALSE THEN
		
		//-----------------------------
		//State Machine
		//-----------------------------
		CASE THIS^.StepNo OF
			MACHINE_RUN_INIT:
				IF THIS^.StepOneShotTrig THEN
					THIS^.Monitoring.StepMessage	:= 'Init: Start.';
					THIS^.Delay(IN:=FALSE);
					Meth_Rest_IO();
				ELSIF Meth_Enable(TRUE) THEN
					THIS^.StepNo	:= 	MACHINE_WAIT_DANCER_FULL;
				//	THIS^.StepNo	:= 	MACHINE_GRIPPER_END_POSITION;
				END_IF								
			
				
			MACHINE_WAIT_DANCER_FULL:
				IF THIS^.StepOneShotTrig THEN
					THIS^.Monitoring.StepMessage	:= 'Wait Dancer full';
					THIS^.Delay(IN:=FALSE);
				ELSIF Meth_WaitDancerFull(TRUE) THEN
					THIS^.StepNo	:= 	MACHINE_GRIPPER_RETRACT;
				END_IF					
								
	
			MACHINE_GRIPPER_RETRACT:
				IF THIS^.StepOneShotTrig THEN
					THIS^.Monitoring.StepMessage	:= 'Gripper retract';
					THIS^.Delay(IN:=FALSE);
					
				ELSIF Meth_gripperRetract(TRUE) THEN
					THIS^.StepNo	:= 	MACHINE_GRIPPER_END_POSITION;
				END_IF	

									
			MACHINE_GRIPPER_END_POSITION:
				IF THIS^.StepOneShotTrig THEN
					THIS^.Monitoring.StepMessage	:= 'Machine WAIT position';
					THIS^.Delay(IN:=FALSE);
				ELSIF Meth_gripperEndPosition(TRUE) THEN
					THIS^.StepNo	:= 	MACHINE_OUT_GRIPPER_START_POSITION;
				END_IF					
			
			MACHINE_OUT_GRIPPER_START_POSITION:
				IF THIS^.StepOneShotTrig THEN
					THIS^.Monitoring.StepMessage	:= 'Output Grippers to start position';
					Meth_OutGripperStartPos(FALSE) ;
				ELSIF Meth_OutGripperStartPos(TRUE) THEN
					THIS^.StepNo	:= 	MACHINE_OUT_GRIPPER_CLAMP;
				END_IF				
							
				
			MACHINE_OUT_GRIPPER_CLAMP:
				IF THIS^.StepOneShotTrig THEN
					THIS^.Monitoring.StepMessage	:= 'Machine grippers clamp';
					THIS^.Delay(IN:=FALSE);
				ELSIF Meth_OutGripperClamp(TRUE) THEN
					THIS^.StepNo	:= 	MACHINE_GRIPPER_OPEN;
				END_IF	
			

			MACHINE_GRIPPER_OPEN:
				IF THIS^.StepOneShotTrig THEN
					THIS^.Monitoring.StepMessage	:= 'Gripper Open';
					THIS^.Delay(IN:=FALSE);
				ELSIF Meth_gripperOpen(TRUE) THEN
					THIS^.StepNo	:= 	MACHINE_GRIPPER_START_POSITION;
				END_IF					
						
				
			MACHINE_GRIPPER_START_POSITION:
				IF THIS^.StepOneShotTrig THEN
					THIS^.Monitoring.StepMessage	:= 'Machine start position';
					THIS^.Delay(IN:=FALSE);
					
				ELSIF Meth_gripperStartPosition(TRUE) THEN
					THIS^.StepNo	:= 	MACHINE_GRIPPER_EXCTRACT;
				END_IF	
	
			
			MACHINE_GRIPPER_EXCTRACT:
			IF THIS^.StepOneShotTrig THEN
				THIS^.Monitoring.StepMessage	:= 'Gripper Extract';
				THIS^.Delay(IN:=FALSE);
			ELSIF Meth_gripperExtract(TRUE) THEN
				THIS^.StepNo	:= 	MACHINE_GRIPPER_CLOSE;
			END_IF				
				
			MACHINE_GRIPPER_CLOSE:
				IF THIS^.StepOneShotTrig THEN
					THIS^.Monitoring.StepMessage	:= 'Gripper Close';
					THIS^.Delay(IN:=FALSE);
				ELSIF Meth_gripperClose(TRUE) THEN
					THIS^.StepNo	:= 	MACHINE_COLD_CUT_VALVE_OPEN;
				END_IF	
	
			MACHINE_COLD_CUT_VALVE_OPEN:
				IF THIS^.StepOneShotTrig THEN
					THIS^.Monitoring.StepMessage	:= 'Cold cut valve open';
					THIS^.Delay(IN:=FALSE);
				ELSIF Meth_ColdCutValveOpen(TRUE) THEN
					THIS^.StepNo	:= 	MACHINE_WELD_VALVE_OPEN;
				END_IF	

			MACHINE_WELD_VALVE_OPEN://and gripper open
				IF THIS^.StepOneShotTrig THEN
					THIS^.Monitoring.StepMessage	:= 'Hot weld valve open press Down';
					THIS^.Delay(IN:=FALSE);
				ELSIF Meth_HotWeldValveOpen(TRUE) THEN
					THIS^.StepNo	:= 	MACHINE_HEATER_ON;
				END_IF					
				
			MACHINE_HEATER_ON://
				IF THIS^.StepOneShotTrig THEN
					THIS^.Monitoring.StepMessage	:= 'Heater ON';
					THIS^.Delay(IN:=FALSE);
				ELSIF Meth_HeaterON(TRUE) THEN
					THIS^.StepNo	:= 	MACHINE_HEATER_OFF;
				END_IF								
				
			MACHINE_HEATER_OFF://gripper retract
				IF THIS^.StepOneShotTrig THEN
					THIS^.Monitoring.StepMessage	:= 'Heater Off';
					THIS^.Delay(IN:=FALSE);
				ELSIF Meth_HeaterOff(TRUE) THEN
					THIS^.StepNo	:= 	MACHINE_CUT_WEB;
				END_IF					
						
			MACHINE_CUT_WEB:
				IF THIS^.StepOneShotTrig THEN
					THIS^.Monitoring.StepMessage	:= 'Close valves';
					THIS^.Delay(IN:=FALSE);
					gMachineCtrl.IO.Out.KniveCut:=NOT(gMachineCtrl.IO.Out.KniveCut);
				ELSIF Meth_CutWeb(TRUE) THEN
					THIS^.StepNo	:= 	MACHINE_VALVE_CLOSE;
				END_IF		
				
			MACHINE_VALVE_CLOSE:
				IF THIS^.StepOneShotTrig THEN
					THIS^.Monitoring.StepMessage	:= 'Close valves';
					THIS^.Delay(IN:=FALSE);
				ELSIF Meth_HeaterValvesClose(TRUE) THEN
					THIS^.StepNo	:= 	MACHINE_OUT_GRIPPER_END_POSITION;
				END_IF					
				
			MACHINE_OUT_GRIPPER_END_POSITION:
				IF THIS^.StepOneShotTrig THEN
					THIS^.Monitoring.StepMessage	:= 'Output Grippers to start position';
					Meth_OutGripperEndPos(FALSE) ;
				ELSIF Meth_OutGripperEndPos(TRUE) THEN
					THIS^.StepNo	:= 	MACHINE_DONE;
				END_IF								
				
			MACHINE_DONE:
				IF THIS^.StepOneShotTrig THEN
					THIS^.Monitoring.StepMessage	:= 'Machine cycle Done';
				ELSIF Meth_Done(TRUE) THEN
					THIS^.StepNo	:= 	MACHINE_RUN_INIT;
				END_IF			
			
				
			//UnUsed	
			
								
		END_CASE
	
	ELSE
		THIS^.Monitoring.StepMessage:= 'Pause';
		
		IF THIS^.Status.Fault = TRUE THEN
		//IF Meth_EmStop(TRUE) THEN
				THIS^.CMD.ResetCycle	:= TRUE;		// Reset the all state machine to start point
		//END_IF
			
		END_IF
		
	END_IF
	
	//============================================================================================
	// Reset Internal Function Blocks
	IF THIS^.CMD.ResetCycle = TRUE THEN
		IF FB_RW_Ctrl_ref.Running OR FB_RW_Ctrl_ref.Pause OR FB_RW_Ctrl_ref.Fault THEN
			FB_RW_Ctrl_ref.ResetCycle	:= TRUE;
		END_IF
	END_IF	
	
	THIS^.FB_HeaterProtection();
	THIS^.Delay();
	THIS^.CH_Logic();
	
	// Reset Meth_EmStop when at Init State
	IF THIS^.Pause = FALSE THEN
		//Meth_EmStop(FALSE);
	END_IF

METHOD PRIVATE Meth_ColdCutValveOpen : BOOL
VAR_INPUT
	Execute: 	BOOL;
END_VAR


	THIS^.Monitoring.StepMessage			:= 'Cold Cut Valve Open';
	THIS^.Monitoring.Error_Text				:= ' Fail';
	//THIS^.CMD.Deacivate_Sequence_Time_Out	:= TRUE;	// Disable time out to the all sequence
	THIS^.CMD.DeactivateStepTimeOut			:= TRUE;	// Disable time out to the actual step
	THIS^.Parameter.TimeOut					:= T#5S;


	
	gMachineCtrl.IO.Out.Buzzer	:=TRUE;
										
	THIS^.Delay.IN:=TRUE;
	THIS^.Delay.PT :=DINT_TO_TIME( Persist.PersistentStruct.TimeColdCutPressDown);// Ctrl_ref.Parameters.TimerPressDown1);
	IF THIS^.Delay.Q THEN
		Meth_ColdCutValveOpen	:= TRUE;
		gMachineCtrl.IO.Out.GripperOpen:=TRUE;
	END_IF
END_METHOD

METHOD Meth_CutWeb : BOOL
VAR_INPUT
	Execute: 	BOOL;
END_VAR
	THIS^.Monitoring.StepMessage			:= 'Cut Web';
	THIS^.Monitoring.Error_Text				:= ' Fail';
	//THIS^.CMD.Deacivate_Sequence_Time_Out	:= TRUE;	// Disable time out to the all sequence
	THIS^.CMD.DeactivateStepTimeOut			:= TRUE;	// Disable time out to the actual step
	THIS^.Parameter.TimeOut					:= T#5S;

	
											
	THIS^.Delay.IN:=TRUE;
	THIS^.Delay.PT :=DINT_TO_TIME( Persist.PersistentStruct.TimeKniveVut);// Ctrl_ref.Parameters.TimerPressDown1);
	IF THIS^.Delay.Q THEN
		Meth_CutWeb	:= TRUE;
		
		//gMachineCtrl.Parameters.UW_1_Param.EnableTension:=TRUE;
		//gMachineCtrl.Parameters.UW_2_Param.EnableTension:=TRUE;
		
	END_IF
END_METHOD

METHOD PRIVATE Meth_Done : BOOL
VAR_INPUT
	Execute: 	BOOL;
END_VAR


	//THIS^.Monitoring.StepMessage			:= 'Press 1 engage';
	//THIS^.Monitoring.Error_Text				:= 'Press 1 engage Fail';
	//THIS^.CMD.Deacivate_Sequence_Time_Out	:= TRUE;	// Disable time out to the all sequence
	//THIS^.CMD.DeactivateStepTimeOut			:= TRUE;	// Disable time out to the actual step
	//THIS^.Parameter.TimeOut					:= T#5S;

	//gMachineCtrl.Parameters.UW_1_Param.EnableDancer :=FALSE;
	//gMachineCtrl.Parameters.UW_2_Param.EnableDancer:=FALSE;	
	
	THIS^.Status.Done		:= TRUE;
	THIS^.Status.Running	:= FALSE;									
	Meth_Done	:= TRUE;
END_METHOD

METHOD PRIVATE Meth_Enable : BOOL
VAR_INPUT
	Execute: 	BOOL;
END_VAR


IF THIS^.CMD.Start THEN
	
	THIS^.Monitoring.StepMessage			:= 'Start';
	THIS^.Monitoring.Error_Text				:= 'Start Fail';
	THIS^.CMD.Deacivate_Sequence_Time_Out	:= TRUE;	// Disable time out to the all sequence
	THIS^.CMD.DeactivateStepTimeOut			:= TRUE;	// Disable time out to the actual step
	THIS^.Parameter.TimeOut					:= T#0.5S;

	THIS^.CMD.Start			:= FALSE;
	THIS^.Status.Done		:= FALSE;
	THIS^.Status.Running	:= TRUE;
	
	// Reset Commands and Statuses												
	
	Meth_Enable	:= TRUE;
END_IF
END_METHOD

METHOD PRIVATE Meth_gripperClose : BOOL
VAR_INPUT
	Execute: 	BOOL;
END_VAR


	THIS^.Monitoring.StepMessage			:= 'Gripper Close';
	THIS^.Monitoring.Error_Text				:= ' Fail';
	//THIS^.CMD.Deacivate_Sequence_Time_Out	:= TRUE;	// Disable time out to the all sequence
	THIS^.CMD.DeactivateStepTimeOut			:= TRUE;	// Disable time out to the actual step
	THIS^.Parameter.TimeOut					:= T#5S;

	gMachineCtrl.IO.Out.GripperOpen:=TRUE;
											
	THIS^.Delay.IN:=TRUE;
	THIS^.Delay.PT :=DINT_TO_TIME( Persist.PersistentStruct.TimeGripperOpen);// Ctrl_ref.Parameters.TimerPressDown1);
	IF THIS^.Delay.Q THEN
		Meth_gripperClose	:= TRUE;
		
		//gMachineCtrl.Parameters.UW_1_Param.EnableTension:=TRUE;
		//gMachineCtrl.Parameters.UW_2_Param.EnableTension:=TRUE;
		
	END_IF
END_METHOD

METHOD PRIVATE Meth_gripperEndPosition : BOOL
VAR_INPUT
	Execute: 	BOOL;
END_VAR


	//THIS^.Monitoring.StepMessage			:= 'GripperStartPosition';
	THIS^.Monitoring.Error_Text				:= ' Fail';
	//THIS^.CMD.Deacivate_Sequence_Time_Out	:= TRUE;	// Disable time out to the all sequence
	THIS^.CMD.DeactivateStepTimeOut			:= TRUE;	// Disable time out to the actual step
	THIS^.Parameter.TimeOut					:= T#5S;

	gMachineCtrl.IO.Out.GripperPistonPosition:=TRUE;
	
	gMachineCtrl.IO.Out.ExternalNipMotor:=TRUE;
		
	//gMachineCtrl.Parameters.UW_1_Param.kp := gMachineCtrl.Parameters.UW_1_Param.kpMove;
	////gMachineCtrl.Parameters.UW_1_Param.TN := gMachineCtrl.Parameters.UW_1_Param.TNMove;
	//.Parameters.UW_2_Param.kp := gMachineCtrl.Parameters.UW_2_Param.kpMove;
	//gMachineCtrl.Parameters.UW_2_Param.TN := gMachineCtrl.Parameters.UW_2_Param.TNMove;



							
	THIS^.Delay.IN:=TRUE;
	THIS^.Delay.PT :=DINT_TO_TIME( Persist.PersistentStruct.TimeGripperStartPosition);// Ctrl_ref.Parameters.TimerPressDown1);
	IF THIS^.Delay.Q THEN
		Meth_gripperEndPosition	:= TRUE;
		
	//.Parameters.UW_1_Param.kp := 0.1;
	//gMachineCtrl.Parameters.UW_1_Param.TN := T#0MS;
	//gMachineCtrl.Parameters.UW_2_Param.kp := 0.1;
	//gMachineCtrl.Parameters.UW_2_Param.TN := T#0MS;			
	
	gMachineCtrl.IO.Out.ExternalNipMotor:=FALSE;
		
	END_IF
END_METHOD

METHOD PRIVATE Meth_gripperExtract : BOOL
VAR_INPUT
	Execute: 	BOOL;
END_VAR


	//THIS^.Monitoring.StepMessage			:= 'Gripper Retract';
	THIS^.Monitoring.Error_Text				:= ' Fail';
	//THIS^.CMD.Deacivate_Sequence_Time_Out	:= TRUE;	// Disable time out to the all sequence
	THIS^.CMD.DeactivateStepTimeOut			:= TRUE;	// Disable time out to the actual step
	THIS^.Parameter.TimeOut					:= T#5S;

	gMachineCtrl.IO.Out.GripperRetract:=TRUE;
											
	THIS^.Delay.IN:=TRUE;
	THIS^.Delay.PT :=DINT_TO_TIME( Persist.PersistentStruct.TimeGripperRetract);// Ctrl_ref.Parameters.TimerPressDown1);
	IF THIS^.Delay.Q THEN
		Meth_gripperExtract	:= TRUE;
	END_IF
END_METHOD

METHOD PRIVATE Meth_gripperOpen : BOOL
VAR_INPUT
	Execute: 	BOOL;
END_VAR


	//THIS^.Monitoring.StepMessage			:= 'Gripper Open';
	THIS^.Monitoring.Error_Text				:= ' Fail';
	//THIS^.CMD.Deacivate_Sequence_Time_Out	:= TRUE;	// Disable time out to the all sequence
	THIS^.CMD.DeactivateStepTimeOut			:= TRUE;	// Disable time out to the actual step
	THIS^.Parameter.TimeOut					:= T#5S;

	gMachineCtrl.IO.Out.GripperOpen:=FALSE;
											
	THIS^.Delay.IN:=TRUE;
	THIS^.Delay.PT :=DINT_TO_TIME( Persist.PersistentStruct.TimeGripperOpen);// Ctrl_ref.Parameters.TimerPressDown1);
	IF THIS^.Delay.Q THEN
		Meth_gripperOpen	:= TRUE;
	END_IF
END_METHOD

METHOD PRIVATE Meth_gripperRetract : BOOL
VAR_INPUT
	Execute: 	BOOL;
END_VAR


	//THIS^.Monitoring.StepMessage			:= 'Gripper Retract';
	THIS^.Monitoring.Error_Text				:= ' Fail';
	//THIS^.CMD.Deacivate_Sequence_Time_Out	:= TRUE;	// Disable time out to the all sequence
	THIS^.CMD.DeactivateStepTimeOut			:= TRUE;	// Disable time out to the actual step
	THIS^.Parameter.TimeOut					:= T#5S;

	gMachineCtrl.IO.Out.GripperRetract:=FALSE;
											
	THIS^.Delay.IN:=TRUE;
	THIS^.Delay.PT :=DINT_TO_TIME( Persist.PersistentStruct.TimeGripperRetract);// Ctrl_ref.Parameters.TimerPressDown1);
	IF THIS^.Delay.Q THEN
		Meth_gripperRetract	:= TRUE;
	END_IF
END_METHOD

METHOD PRIVATE Meth_gripperStartPosition : BOOL
VAR_INPUT
	Execute: 	BOOL;
END_VAR


	//THIS^.Monitoring.StepMessage			:= 'GripperStartPosition';
	THIS^.Monitoring.Error_Text				:= ' Fail';
	//THIS^.CMD.Deacivate_Sequence_Time_Out	:= TRUE;	// Disable time out to the all sequence
	THIS^.CMD.DeactivateStepTimeOut			:= TRUE;	// Disable time out to the actual step
	THIS^.Parameter.TimeOut					:= T#5S;

	gMachineCtrl.IO.Out.GripperPistonPosition:=FALSE;
											
	THIS^.Delay.IN:=TRUE;
	THIS^.Delay.PT :=DINT_TO_TIME( Persist.PersistentStruct.TimeGripperHomePosition);// Ctrl_ref.Parameters.TimerPressDown1);
	IF THIS^.Delay.Q THEN
		Meth_gripperStartPosition	:= TRUE;
	END_IF
END_METHOD

METHOD PRIVATE Meth_HeaterOff : BOOL
VAR_INPUT
	Execute: 	BOOL;
END_VAR


	THIS^.Monitoring.StepMessage			:= 'Heater Off';
	THIS^.Monitoring.Error_Text				:= ' Heater Off Fail';
	//THIS^.CMD.Deacivate_Sequence_Time_Out	:= TRUE;	// Disable time out to the all sequence
	THIS^.CMD.DeactivateStepTimeOut			:= TRUE;	// Disable time out to the actual step
	THIS^.Parameter.TimeOut					:= T#5S;

	
											
	THIS^.Delay.IN:=TRUE;
	THIS^.Delay.PT :=DINT_TO_TIME( Persist.PersistentStruct.TimerHotWeldingOff);// Ctrl_ref.Parameters.TimerPressDown1);
	IF THIS^.Delay.Q AND THIS^.FB_HeaterProtection.Done THEN
		Meth_HeaterOff	:= TRUE;
	END_IF
END_METHOD

METHOD PRIVATE Meth_HeaterON : BOOL
VAR_INPUT
	Execute: 	BOOL;
END_VAR


	THIS^.Monitoring.StepMessage			:= 'Heater ON';
	THIS^.Monitoring.Error_Text				:= ' Heater ON Fail';
	//THIS^.CMD.Deacivate_Sequence_Time_Out	:= TRUE;	// Disable time out to the all sequence
	THIS^.CMD.DeactivateStepTimeOut			:= TRUE;	// Disable time out to the actual step
	THIS^.Parameter.TimeOut					:= T#5S;

	//Ctrl_ref.IO.Out.HeaterOn := TRUE;
	FB_HeaterProtection.Excute:=TRUE;
			
	gMachineCtrl.IO.Out.ColdCutPistonDown:=TRUE;						
//	THIS^.Delay.IN:=TRUE;
//	THIS^.Delay.PT :=DINT_TO_TIME( Persist.PersistentStruct.TimerHotWeldingOn);// Ctrl_ref.Parameters.TimerPressDown1);
//	IF THIS^.Delay.Q THEN
		Meth_HeaterON	:= TRUE;;
//	END_IF
END_METHOD

METHOD PRIVATE Meth_HeaterValvesClose : BOOL
VAR_INPUT
	Execute: 	BOOL;
END_VAR


	THIS^.Monitoring.StepMessage			:= 'Valves close';
	THIS^.Monitoring.Error_Text				:= ' Valves close Fail';
	//THIS^.CMD.Deacivate_Sequence_Time_Out	:= TRUE;	// Disable time out to the all sequence
	THIS^.CMD.DeactivateStepTimeOut			:= TRUE;	// Disable time out to the actual step
	THIS^.Parameter.TimeOut					:= T#5S;

	gMachineCtrl.IO.Out.PressDown:=FALSE;
	gMachineCtrl.IO.Out.ColdCutPistonDown:=FALSE;										
	THIS^.Delay.IN:=TRUE;
	THIS^.Delay.PT :=DINT_TO_TIME( Persist.PersistentStruct.TimerPressUp);// Ctrl_ref.Parameters.TimerPressDown1);
	IF THIS^.Delay.Q THEN
		Meth_HeaterValvesClose	:= TRUE;
	END_IF
END_METHOD

METHOD PRIVATE Meth_HotWeldValveOpen : BOOL
VAR_INPUT
	Execute: 	BOOL;
END_VAR


	THIS^.Monitoring.StepMessage			:= 'Hot Weld Valve Open';
	THIS^.Monitoring.Error_Text				:= ' Hot Weld Valve Open Fail';
	//THIS^.CMD.Deacivate_Sequence_Time_Out	:= TRUE;	// Disable time out to the all sequence
	THIS^.CMD.DeactivateStepTimeOut			:= TRUE;	// Disable time out to the actual step
	THIS^.Parameter.TimeOut					:= T#5S;

	gMachineCtrl.IO.Out.PressDown :=TRUE;
											
	THIS^.Delay.IN:=TRUE;
	THIS^.Delay.PT :=DINT_TO_TIME( Persist.PersistentStruct.TimeHotWeldPressDown);// Ctrl_ref.Parameters.TimerPressDown1);
	IF THIS^.Delay.Q THEN
		Meth_HotWeldValveOpen	:= TRUE;
		gMachineCtrl.IO.Out.Buzzer	:=FALSE;
	END_IF
END_METHOD

METHOD Meth_Init :BOOL
VAR_INPUT
END_VAR
Meth_Init:=TRUE;
END_METHOD

